METHOD M_AddChild : ERRORID
VAR_INPUT
	pObject : POINTER TO FB_Object;
	nSlotNr	: UINT;
	nIndex 	: INT;
END_VAR
//Der Delodot-Dispenser kann folgende Objekt-Typen aufnehmen
//Camera, Exposure, Nozzle
IF pObject > 0 THEN
	IF pObject^.P_eObjectType = E_ObjectType.OBJECTTYPE_Camera OR
		pObject^.P_eObjectType = E_ObjectType.OBJECTTYPE_Exposure OR
		pObject^.P_eObjectType = E_ObjectType.OBJECTTYPE_DummyTool OR
		pObject^.P_eObjectType = E_ObjectType.OBJECTTYPE_Nozzle THEN
		M_AddChild := SUPER^.M_AddChild(pObject,nSlotNr,nIndex);
	ELSE
		M_AddChild := E_ErrorIdObjMgmt.ERRORID_InvalidParentObject;
	END_IF
ELSE
	M_AddChild := E_ErrorIdObjMgmt.ERRORID_InvalidParentObject;
END_IF
END_METHOD

METHOD M_CancelAction
VAR_INPUT
	eAction : E_Action;
END_VAR
CASE eAction OF
	E_Action.ACTION_SetPressure:
		IF bSetPress  THEN
			fbSetPress(bExecute:= FALSE, pPneuChannelRef:= pPneuChannelPress);
		END_IF	
	E_Action.ACTION_SwitchPressure:
		IF bSwitchPress AND nStateA_SwitchPress < 70 THEN
			nStateA_SwitchPress := 70;
		END_IF
	E_Action.ACTION_DispenseDrops:
		IF bDispense AND nStateA_Dispense < 70 THEN
			nStateA_Dispense := 70;
		END_IF
ELSE
	SUPER^.M_CancelAction(eAction);
END_CASE
END_METHOD

METHOD M_CheckAction : ERRORID
VAR_INPUT
	refActionData 	: REFERENCE TO ST_ActionData;
	pCorrelObject	: POINTER TO FB_Object;
END_VAR

VAR
END_VAR
CASE refActionData.eAction OF
	E_Action.ACTION_DispenseDrops, //BasicAction für ActionOnArray
	E_Action.ACTION_TeachTarget:
		RETURN;
ELSE
	M_CheckAction := SUPER^.M_CheckAction(refActionData, pCorrelObject);
END_CASE
END_METHOD

METHOD M_CheckProcDataType : BOOL
VAR_INPUT
	eProcDataType : E_ProcDataType;
END_VAR
IF eProcDataType = E_ProcDataType.PROCDATATYPE_Temp1 THEN
	M_CheckProcDataType := TRUE;
END_IF
END_METHOD

METHOD M_ClearAllProps
VAR_INPUT
	bIgnoreParent : BOOL; //Es wird das gesamte OD gelöscht. -> Zeiger auf Parent nicht mehr gültig!
END_VAR
pPneuChannelPress := 0;
SUPER^.M_ClearAllProps(bIgnoreParent);
END_METHOD

METHOD M_ExeAction : ERRORID
VAR_INPUT
	refActionData : REFERENCE TO ST_ActionData;	
END_VAR
IF NOT (eCurrentState = E_MachineState.MACHINESTATE_Idle OR
	eCurrentState = E_MachineState.MACHINESTATE_Active OR
	eCurrentState = E_MachineState.MACHINESTATE_Ready) THEN
	M_ExeAction := E_ErrorIdCmd.ERRORID_InvalidState;
	RETURN;
END_IF

CASE refActionData.eAction OF
	
	E_Action.ACTION_Init:
		IF NOT bInitAxis AND NOT bInitTool THEN
			bInitAxis := TRUE;
			bInitTool := TRUE;
			fbList.A_AddHeadValue(hList:= hList, putValue := E_Action.ACTION_Init);	//InitAxis
			fbList.A_AddHeadValue(hList:= hList, putValue := E_Action.ACTION_Init);	//InitTool
		ELSE
			RETURN;
		END_IF
		
	E_Action.ACTION_SetPressure:
		fbSetPress(bExecute:= FALSE, pPneuChannelRef:= pPneuChannelPress); //eventueller Fehler wird auch zurückgesetzt
		fbSetPress.bAwait := DINT_TO_BOOL(refActionData.aParams[1]);
		fbSetPress.nValue := DINT_TO_INT(refActionData.aParams[2]);
		fbSetPress.nTolerancePlus := DINT_TO_INT(refActionData.aParams[3]);
		fbSetPress.nToleranceMinus := DINT_TO_INT(refActionData.aParams[4]);
		fbSetPress.tTimeout := DINT_TO_TIME(refActionData.aParams[5]);
		
		fbSetPress(bExecute:= TRUE,	pPneuChannelRef:= pPneuChannelPress,nErrorId=> M_ExeAction);
		IF fbSetPress.bError THEN
			RETURN;
		END_IF
		
		IF NOT bSetPress AND fbSetPress.bBusy THEN
			bSetPress := TRUE;
			fbList.A_AddHeadValue(hList := hList, putValue := E_Action.ACTION_SetPressure);
		ELSE
			RETURN;	
		END_IF

	E_Action.ACTION_SwitchPressure:
		eSwitchPressCtrl := DINT_TO_USINT(refActionData.aParams[1]);
		IF (eSwitchPressCtrl = E_PressCtrl.PRESSCTRL_PressOn) OR (eSwitchPressCtrl = E_PressCtrl.PRESSCTRL_Off) THEN
			tPressTime := DINT_TO_TIME(refActionData.aParams[2]);
			//Wenn Aktion aktiv kann es sein das die Zeit noch läuft oder der Druck an ist
			IF bSwitchPress THEN	//Aktion ist aktiv
				IF eSwitchPressCtrl = E_PressCtrl.PRESSCTRL_PressOn THEN
					//Statemachine zurücksetzen
					nStateA_SwitchPress := 0;		
				ELSE
					pFbMultiZ^.M_SetDigiOut(nChannel:= nDOutChanValvePress, bValue:= FALSE);
					nStateA_SwitchPress := 80;
				END_IF
			ELSE	//Aktion ist nicht aktiv
				IF eSwitchPressCtrl = E_PressCtrl.PRESSCTRL_PressOn THEN
					bSwitchPress := TRUE;
					fbList.A_AddHeadValue(hList := hList, putValue := E_Action.ACTION_SwitchPressure);
				ELSE
					pFbMultiZ^.M_SetDigiOut(nChannel:= nDOutChanValvePress, bValue:= FALSE);
				END_IF
			END_IF
		ELSE
			M_ExeAction := E_ErrorIdCmd.ERRORID_InvalidCtrl;
			RETURN;
		END_IF		
		
	E_Action.ACTION_DispenseDrops:
		bDispenseStart := DINT_TO_BOOL(refActionData.aParams[2]);
		IF NOT bDispense AND bDispenseStart THEN
			nDrops := DINT_TO_UINT(refActionData.aParams[1]);
			fbList.A_AddHeadValue( hList := hList, putValue := E_Action.ACTION_DispenseDrops);
			bDispense := TRUE;
		ELSE
			pTripleTrigRef^.M_TriggerOff(nTriggerChannel);
		END_IF

	ELSE
		M_ExeAction := SUPER^.M_ExeAction(refActionData);
		RETURN;
END_CASE
bBusy := TRUE;
eCurrentState := E_MachineState.MACHINESTATE_Active;
END_METHOD

METHOD M_GetAllProps : ERRORID
VAR_INPUT
	refCmdData : REFERENCE TO  ST_CmdData;
END_VAR
//BaseProperties lesen
SUPER^.M_GetAllProps(refCmdData);
//BaseProperties lesen
nCurrentPropIndex := nCurrentPropIndex + 1; //SubType (Reserve)
refCmdData.n32Data[nCurrentPropIndex] := nSubType;
nCurrentPropIndex := nCurrentPropIndex + 1;
refCmdData.n32Data[nCurrentPropIndex] := nTriggerChannel;
IF pTripleTrigRef > 0 THEN
	nCurrentPropIndex := nCurrentPropIndex + 1;
	refCmdData.n32Data[nCurrentPropIndex] := pTripleTrigRef^.M_GetFrequency(nTriggerChannel);
	nCurrentPropIndex := nCurrentPropIndex + 1;
	refCmdData.n32Data[nCurrentPropIndex] := pTripleTrigRef^.M_GetPulse(nTriggerChannel);
	nCurrentPropIndex := nCurrentPropIndex + 1;
	refCmdData.n32Data[nCurrentPropIndex] := pTripleTrigRef^.M_GetAmplitudePercent(nTriggerChannel);
ELSE
	nCurrentPropIndex := nCurrentPropIndex + 3;
END_IF
nCurrentPropIndex := nCurrentPropIndex + 1;
IF pPneuChannelPress > 0 THEN
	refCmdData.n32Data[nCurrentPropIndex] := pPneuChannelPress^.nChannel;
ELSE
	refCmdData.n32Data[nCurrentPropIndex] := 0;
END_IF
nCurrentPropIndex := nCurrentPropIndex + 1; 
refCmdData.n32Data[nCurrentPropIndex] := nDOutChanValvePress; //Digitaler Ausgangskanal MzHead Druckventil
END_METHOD

METHOD M_SetAllProps : ERRORID
VAR_INPUT
	refCmdData : REFERENCE TO  ST_CmdData;
END_VAR

VAR
	nPneuChannel : USINT;
END_VAR
M_SetAllProps := SUPER^.M_SetAllProps(refCmdData);

IF M_SetAllProps > 0 THEN
	RETURN;
END_IF

{IF defined (variable:aFbTripleTriggerRef)}
pTripleTrigRef := ADR(aFbTripleTriggerRef[1]);
{ELSE}
M_SetAllProps := E_ErrorIdObjMgmt.ERRORID_InvalidHardwareRef;
RETURN;
{END_IF}

//SubType (Reserve)
nCurrentPropIndex := nCurrentPropIndex + 1;
nSubType := refCmdData.n32Data[nCurrentPropIndex];
//TriggerChannel
nCurrentPropIndex := nCurrentPropIndex + 1;
nSpecPropIndex := nCurrentPropIndex;
nTriggerChannel := DINT_TO_USINT(refCmdData.n32Data[nCurrentPropIndex]);
IF NOT (nTriggerChannel >= 1 AND nTriggerChannel <= 3) THEN
	M_SetAllProps := E_ErrorIdObjMgmt.ERRORID_InvalidTriggerChannel;
	RETURN;
END_IF

//Frequenz
nCurrentPropIndex := nCurrentPropIndex + 1;
IF NOT (refCmdData.n32Data[nCurrentPropIndex] >= 16 AND refCmdData.n32Data[nCurrentPropIndex] <= 1000000) THEN	
	M_SetAllProps := E_ErrorIdObjMgmt.ERRORID_InvalidFrequency;
	RETURN;
END_IF
pTripleTrigRef^.M_SetFrequency(nTriggerChannel,refCmdData.n32Data[nCurrentPropIndex]);

//Plusbreite
nCurrentPropIndex := nCurrentPropIndex + 1;
IF NOT (refCmdData.n32Data[nCurrentPropIndex] >= 0 AND refCmdData.n32Data[nCurrentPropIndex] <= 65535) THEN
	M_SetAllProps := E_ErrorIdObjMgmt.ERRORID_InvalidPulseWidth;  //Error
	RETURN;
END_IF
pTripleTrigRef^.M_SetPulse(nTriggerChannel,DINT_TO_UINT(refCmdData.n32Data[nCurrentPropIndex]));

//Stroke(Hub) in % (1 Stelle hinter Komma)
nCurrentPropIndex := nCurrentPropIndex + 1;
IF NOT (refCmdData.n32Data[nCurrentPropIndex] >= 0 AND refCmdData.n32Data[nCurrentPropIndex] <= 1000) THEN
	M_SetAllProps := E_ErrorIdObjMgmt.ERRORID_InvalidVoltage;  //Error
	RETURN;
END_IF
pTripleTrigRef^.M_SetAmplitudePercent(nTriggerChannel,DINT_TO_UINT(refCmdData.n32Data[nCurrentPropIndex]));

//PneuChannel Druck
nCurrentPropIndex := nCurrentPropIndex + 1;
nPneuChannel := DINT_TO_USINT(refCmdData.n32Data[nCurrentPropIndex]);
IF NOT (nPneuChannel >= 0 AND nPneuChannel <= cNoOfPneuChannels) THEN
	M_SetAllProps := E_ErrorIdObjMgmt.ERRORID_InvalidPneuChannel;
	RETURN;	
END_IF
pPneuChannelPress := ADR(aFbPneuChannel[nPneuChannel]);

//Digitale Ausgänge auf MzHead müssen zwischen 1 und 7 liegen
nCurrentPropIndex := nCurrentPropIndex + 1;
nDOutChanValvePress := DINT_TO_USINT(refCmdData.n32Data[nCurrentPropIndex]);	//Digitaler Ausgangskanal MzHead Druckventil
IF NOT (nDOutChanValvePress >= 0 AND nDOutChanValvePress <= 7) THEN
	M_SetAllProps := E_ErrorIdObjMgmt.ERRORID_InvalidMzDOutChannel;
	RETURN;	
END_IF

nNoOfProps := nCurrentPropIndex + 1;
END_METHOD

METHOD M_SetSingleProp : ERRORID
VAR_INPUT
	refCmdData : REFERENCE TO  ST_CmdData;
END_VAR
IF nSpecPropIndex = refCmdData.aHeader[1] THEN
	IF refCmdData.n32Data[0] >= 1 AND refCmdData.n32Data[0] <= 3 THEN
		nTriggerChannel := DINT_TO_USINT(refCmdData.n32Data[0]);
	ELSE
		M_SetSingleProp := E_ErrorIdObjMgmt.ERRORID_InvalidTriggerChannel;
		RETURN;
	END_IF
ELSIF (nSpecPropIndex + 1) = refCmdData.aHeader[1] THEN	//Frequenz
	IF NOT (refCmdData.n32Data[0] > 16 AND refCmdData.n32Data[0] < 1000000) THEN
		M_SetSingleProp := E_ErrorIdObjMgmt.ERRORID_InvalidFrequency;
		RETURN;
	END_IF
	pTripleTrigRef^.M_SetFrequency(nTriggerChannel,refCmdData.n32Data[0]);
ELSIF (nSpecPropIndex + 2) = refCmdData.aHeader[1] THEN //Pulsbreite
	IF NOT (refCmdData.n32Data[0] >= 0 AND refCmdData.n32Data[0] < 65535) THEN
		M_SetSingleProp := E_ErrorIdObjMgmt.ERRORID_InvalidPulseWidth;
		RETURN;
	END_IF
	pTripleTrigRef^.M_SetPulse(nTriggerChannel,DINT_TO_UINT(refCmdData.n32Data[0]));
ELSIF (nSpecPropIndex + 3) = refCmdData.aHeader[1] THEN	//Stroke(Hub) in % (1 Stelle hinter Komma)
	IF NOT (refCmdData.n32Data[0] >= 0 AND refCmdData.n32Data[0] <= 1000) THEN
		M_SetSingleProp := E_ErrorIdObjMgmt.ERRORID_InvalidVoltage;
		RETURN;
	END_IF
	pTripleTrigRef^.M_SetAmplitudePercent(nTriggerChannel,DINT_TO_UINT(refCmdData.n32Data[0]));
ELSE
	M_SetSingleProp := SUPER^.M_SetSingleProp(refCmdData);
END_IF
END_METHOD

END_FUNCTION_BLOCK

// ---- Objects/Tools/FB_TriplePip.TcPOU
FUNCTION_BLOCK FB_TriplePip EXTENDS FB_MzTool
VAR_INPUT
END_VAR
VAR_OUTPUT
END_VAR
VAR
	bTipEjectorExist	: BOOL;	

	//SpecProperties
	nDiluterObjId		: UINT;
	pDiluter			: POINTER TO FB_Diluter;
	
	pPneuChannelSynthGas: POINTER TO FB_PneuChannelRef;
	pPneuChannelVac		: POINTER TO FB_PneuChannelRef;
	
	nValveNrSynthGas	: USINT;
	nValveNrVacuum		: USINT;
	nHoldVacuumVial		: INT;
	nHoldVacuumSeptum	: INT;
	rDockOffset			: REAL;
	rXMoveDockFlipTube	: REAL;
	rZMoveDockFlipTube	: REAL;

	//****************************************Aktionvariablen****************************************************
	
	stActionDataSpec	: ST_ActionData;
	
	//Action: "InitSpec"
	bInitSpec			: BOOL;
	bInitSpecFlag		: BOOL := TRUE;
	nStateA_InitSpec	: USINT;
	
	//Action: "Dispense"
	bDispense			: BOOL;
	nStateA_Dispense	: USINT;
	nQuantity			: DINT;
	nFlow				: DINT;
	
	//Action: "SetPressure"
	bSetPress			: BOOL;
	fbSetPress			: FB_SetPressure;

	//Action: "SetVacuum"
	bSetVacuum			: BOOL;
	fbSetVacuum			: FB_SetPressure;
	
	//Action: "SwitchPressure"
	bSwitchPress		: BOOL;			
	nStateA_SwitchPress	: USINT;		//State von A_SwitchPress()
	nSwitchPressChannel	: USINT;
	eSwitchPressCtrl	: E_PressCtrl;
	tPressTime			: TIME;			//nach dieser Zeit Ventil automatisch wieder zu
	timerPress			: TON;			//Timer für Öffnungszeit Druckventil 		
	
END_VAR

IF eCurrentState = E_MachineState.MACHINESTATE_Active THEN
	IF bInitSpec THEN
		A_InitSpec();
		IF nStateA_InitSpec >= 80 THEN
			IF nStateA_InitSpec >= 99 THEN
				bError := TRUE;		
			END_IF
			bInitSpec := FALSE;
			nStateA_InitSpec := 0;
			M_RemoveListEntry(nSearchValue:= E_Action.ACTION_Init);
		END_IF		
	END_IF
	
	IF bDispense THEN
		A_Dispense();
		IF nStateA_Dispense >= 80 THEN
			IF nStateA_Dispense >= 99 THEN
				bError := TRUE;	
			END_IF
			bDispense := FALSE;
			nStateA_Dispense := 0;
			M_RemoveListEntry(nSearchValue:= E_Action.ACTION_Dispense);
		END_IF
	END_IF
	
	IF bSetPress THEN
		fbSetPress(pPneuChannelRef:= pPneuChannelSynthGas);
		IF NOT fbSetPress.bBusy THEN
			IF fbSetPress.bError THEN
				bError := TRUE;
				stError.ErrorId := fbSetPress.nErrorId;
				stError.POU := E_POU.POU_FB_TriplePip;
				fbErrorList.M_Add(stError);
			END_IF
			bSetPress := FALSE;
			fbSetPress(pPneuChannelRef:= pPneuChannelSynthGas, bExecute:= FALSE);
			M_RemoveListEntry(nSearchValue:= E_Action.ACTION_SetPressure);
		END_IF
	END_IF	

	IF bSetVacuum THEN
		fbSetVacuum(pPneuChannelRef:= pPneuChannelVac);
		IF NOT fbSetVacuum.bBusy THEN
			IF fbSetVacuum.bError THEN
				bError := TRUE;
				stError.ErrorId := fbSetVacuum.nErrorId;
				stError.POU := E_POU.POU_FB_TriplePip;
				fbErrorList.M_Add(stError);
			END_IF
			bSetVacuum := FALSE;
			fbSetVacuum(pPneuChannelRef:= pPneuChannelVac, bExecute:= FALSE);
			M_RemoveListEntry(nSearchValue:= E_Action.ACTION_SetVacuum);
		END_IF
	END_IF	
	
	IF bSwitchPress THEN	//Kartuschendruck einstellen und Ein-bzw. Aus schalten 
		A_SwitchPress();
		IF nStateA_SwitchPress >= 80 THEN
			IF nStateA_SwitchPress >= 99 THEN
				bError := TRUE;
			END_IF
			bSwitchPress := FALSE;
			nStateA_SwitchPress := 0;
			M_RemoveListEntry(nSearchValue:= E_Action.ACTION_SwitchPressure);
		END_IF
	END_IF	
END_IF

SUPER^();	//FB_MzTool aufrufen

//Prozessdaten aktualisieren
IF pPneuChannelSynthGas > 0 THEN
	stProcessData.n32Data[7] := pPneuChannelSynthGas^.P_nCurrentPressure;
END_IF

IF pPneuChannelVac > 0 THEN
	stProcessData.n32Data[8] := pPneuChannelVac^.P_nCurrentPressure;
END_IF

IF nValveNrSynthGas > 0 THEN
	IF aValves[nValveNrSynthGas].bDigiOut1 THEN
		stProcessData.n32Data[9] := E_PressCtrl.PRESSCTRL_PressOn;
	ELSE
		stProcessData.n32Data[9] := E_PressCtrl.PRESSCTRL_Off;
	END_IF
END_IF

IF nValveNrVacuum > 0 THEN
	IF aValves[nValveNrVacuum].bDigiOut1 THEN
		stProcessData.n32Data[10] := E_PressCtrl.PRESSCTRL_VacOn;
	ELSE
		stProcessData.n32Data[10] := E_PressCtrl.PRESSCTRL_Off;
	END_IF
END_IF

aObjProcData[nNotifyId] := stProcessData;

ACTION A_Dispense:
IF pDiluter^.P_bError THEN
	stError.ErrorId := pDiluter^.P_nErrorId;
	stError.POUState := nStateA_Dispense;
	nStateA_Dispense := 99;
END_IF

CASE nStateA_Dispense OF
	0:	MEMSET(ADR(stActionDataSpec),0,SIZEOF(stActionDataSpec));
		//stActionDataSpec.bIntern := TRUE;
		stActionDataSpec.eAction := E_Action.ACTION_DilPump;
		stActionDataSpec.aParams[1] := E_DilPumpMode.MODE_Press;
		stActionDataSpec.aParams[2] := nQuantity; 
		stActionDataSpec.aParams[3] := nFlow;
		//stActionDataSpec.aParams[4] := 2000; //ReloadSpeed wird von DilConfig übernommen
		//stActionDataSpec.aParams[5] := 1; //Valve-Position für Pump
		//stActionDataSpec.aParams[6] := 2; //Valve-Position für Reload
		
		stError.ErrorId := pDiluter^.M_ExeAction(stActionDataSpec);
		IF stError.ErrorId > 0 THEN
			stError.POUState := nStateA_Dispense;
			nStateA_Dispense := 99;
		ELSE
			nStateA_Dispense := 1;	
		END_IF
		
	1:	//Warten bis Dispensierung fertig
		IF NOT pDiluter^.M_GetActionBusy(E_Action.ACTION_DilPump) THEN
			nStateA_Dispense := 80;
		END_IF
		
	70:	//Abbrechen
		MEMSET(ADR(stActionDataSpec),0,SIZEOF(stActionDataSpec));
		//stActionDataSpec.bIntern := TRUE;
		stActionDataSpec.eAction := E_Action.ACTION_Stop;
		
		pDiluter^.M_ExeAction(stActionDataSpec);
		nStateA_Dispense := 71;
		
	71:	
		IF NOT pDiluter^.P_bBusy THEN
			nStateA_Dispense := 80;
		END_IF
END_CASE

//Errorhandling
IF nStateA_Dispense = 99 THEN
	stError.Cmd := E_Action.ACTION_Dispense;
	stError.POU := E_POU.POU_FB_TriplePip;
	stError.POUAction := E_POUACT.POUACT_A_Dispense;
	fbErrorList.M_Add(stError);
END_IF
END_ACTION

ACTION A_InitSpec:
CASE nStateA_InitSpec OF
	0:	//Checken ob Diluter richtg zugeordnet
		
		IF fbObjectDirectory.M_GetObjType(nDiluterObjId) = E_ObjectType.OBJECTTYPE_Diluter THEN
			nStateA_InitSpec := 80;
		ELSE
			stError.ErrorId := E_ErrorIdObjMgmt.ERRORID_InvalidDiluterObjId;
			nStateA_InitSpec := 99;
		END_IF
	
	1:	//Checken ob notwendige Flüssigleiten vorhanden
	
	2:	//PCV-Level-Controlle aktivieren
	
END_CASE
END_ACTION

ACTION A_Reset:
//Ist noch eine Aktion aktiv?
IF nStateA_ResetSpec = 0 THEN 
	IF bDispense THEN
		bDispense := FALSE;
		nStateA_Dispense := 0;
	END_IF
	
	nStateA_ResetSpec := 80;
END_IF

SUPER^.A_Reset();
END_ACTION

ACTION A_Stop:
IF nStateA_Stop = 0 THEN

	IF bDispense AND nStateA_Dispense < 70 THEN
		nStateA_Dispense := 70;
	END_IF
	
	IF bSetPress THEN
		fbSetPress(bExecute:= FALSE, pPneuChannelRef:= pPneuChannelSynthGas);
	END_IF

	IF bSetVacuum THEN
		fbSetVacuum(bExecute:= FALSE, pPneuChannelRef:= pPneuChannelVac);
	END_IF
		
	
	nStateA_Stop := 1;
END_IF

SUPER^.A_Stop();
END_ACTION

ACTION A_SwitchPress:
CASE nStateA_SwitchPress OF
	0:	//Ventil Einschalten
		IF eSwitchPressCtrl = E_PressCtrl.PRESSCTRL_PressOn OR eSwitchPressCtrl = E_PressCtrl.PRESSCTRL_VacOn THEN
			aValves[M_GetValveNr(nSwitchPressChannel)].M_On(1);
		END_IF
	
		//Timer starten
		IF tPressTime = T#0S THEN
			nStateA_SwitchPress := 80;
			RETURN;	
		END_IF
		
		timerPress(IN:= FALSE);
		timerPress(IN:= TRUE, PT:= tPressTime);
		nStateA_SwitchPress := 1;
		
	1:	//Warten bis Zeitabgelaufen
		timerPress();
		IF timerPress.Q THEN
			timerPress(IN:= FALSE);
			aValves[M_GetValveNr(nSwitchPressChannel)].M_Off();
			nStateA_SwitchPress := 80;
		END_IF
		
	70:	//Abbrechen
		timerPress(IN:= FALSE);
		aValves[M_GetValveNr(nSwitchPressChannel)].M_Off();
		nStateA_SwitchPress := 80;
END_CASE
END_ACTION

METHOD FB_init : BOOL
VAR_INPUT
	bInitRetains : BOOL; // if TRUE, the retain variables are initialized (warm start / cold start)
	bInCopyCode : BOOL;  // if TRUE, the instance afterwards gets moved into the copy code (online change)
END_VAR
eObjectType := E_ObjectType.OBJECTTYPE_TriplePip;
eObjectGroup := E_ObjectGroup.OBJECTGROUP_MzTool OR E_ObjectGroup.OBJECTGROUP_Device;
END_METHOD

METHOD M_AddChild : ERRORID
VAR_INPUT
	pObject : POINTER TO FB_Object;
	nSlotNr	: UINT;
	nIndex 	: INT;
END_VAR
//Kann folgende Objekt-Typen aufnehmen
//Vial
IF pObject > 0 THEN
	IF pObject^.P_eObjectType = E_ObjectType.OBJECTTYPE_Vial THEN
		M_AddChild := SUPER^.M_AddChild(pObject,nSlotNr,nIndex);
	ELSE
		M_AddChild := E_ErrorIdObjMgmt.ERRORID_InvalidParentObject;
	END_IF
ELSE
	M_AddChild := E_ErrorIdObjMgmt.ERRORID_InvalidParentObject;
END_IF
END_METHOD

METHOD M_CancelAction
VAR_INPUT
	eAction : E_Action;
END_VAR
CASE eAction OF
	E_Action.ACTION_Dispense:
		IF bDispense AND nStateA_Dispense < 70 THEN
			nStateA_Dispense := 70;
		END_IF
		
	E_Action.ACTION_SetPressure:
		IF bSetPress THEN
			fbSetPress(bExecute:= FALSE, pPneuChannelRef:= pPneuChannelSynthGas);
		END_IF
	
	E_Action.ACTION_SetVacuum:
		IF bSetVacuum THEN
			fbSetVacuum(bExecute:= FALSE, pPneuChannelRef:= pPneuChannelVac);
		END_IF
		
	E_Action.ACTION_SwitchPressure:
		IF bSwitchPress AND nStateA_SwitchPress < 70 THEN
			nStateA_SwitchPress := 70;
		END_IF	
ELSE
	SUPER^.M_CancelAction(eAction);
END_CASE
END_METHOD

METHOD M_CheckAction : ERRORID
VAR_INPUT
	refActionData 	: REFERENCE TO ST_ActionData;
	pCorrelObject	: POINTER TO FB_Object;
END_VAR

VAR
	pRack : POINTER TO FB_Rack;
	pReactor : POINTER TO FB_Reactor;
	pSlot : POINTER TO FB_PieceSlot;
	pTarget : POINTER TO FB_TargetBase;
END_VAR
CASE refActionData.eAction OF
	E_Action.ACTION_ExchangePiece:
		pTarget := fbObjectDirectory.M_GetObjPointer(refActionData.nTarget);
		//Welches Piece soll gehandelt werden?
		IF refActionData.aParams[2] = 0 THEN //Drop
			IF pPiece = 0 THEN
				M_CheckAction := E_ErrorIdCmd.ERRORID_NoPieceOnTool;
				RETURN;	
			END_IF
			//TripePip kann folgende Pieces handeln
			//Vial, Septum
			IF pPiece^.P_eObjectType = E_ObjectType.OBJECTTYPE_Vial THEN
				//Target muss VialRack oder Reaktor sein
				IF pTarget^.P_eObjectType = E_ObjectType.OBJECTTYPE_VialRack THEN
					pRack := pTarget;
					//Slot muss frei sein
					pSlot := pRack^.M_GetSlot(DINT_TO_UINT(refActionData.aParams[1]));
					IF pSlot = 0 THEN
						M_CheckAction := E_ErrorIdCmd.ERRORID_InvalidTargetSlot;
						RETURN;
					ELSIF pSlot^.P_pPiece > 0 THEN
						M_CheckAction := E_ErrorIdCmd.ERRORID_PieceAlreadyInSlot;
						RETURN;
					END_IF
				ELSIF pTarget^.P_eObjectType = E_ObjectType.OBJECTTYPE_Reactor THEN
					//Slot muss frei sein
					//Hier kann ein Vial geholt werden
					pReactor := pTarget;
					IF pReactor^.P_pVial > 0 THEN
						M_CheckAction := E_ErrorIdCmd.ERRORID_PieceAlreadyInSlot;
						RETURN;
					END_IF
				ELSE
					M_CheckAction := E_ErrorIdCmd.ERRORID_UnsuitableTarget;
					RETURN;
				END_IF
			ELSIF pPiece^.P_eObjectType = E_ObjectType.OBJECTTYPE_Septum THEN
				//Target kann nur Reaktor mit Vial sein
				//Ob ein Vial im Reaktor steht, wird in FB_Reactor.M_CheckActon() geprüft 
				IF pTarget^.P_eObjectType <> E_ObjectType.OBJECTTYPE_Reactor THEN 
					M_CheckAction := E_ErrorIdCmd.ERRORID_UnsuitableTarget;
					RETURN;
				END_IF
			ELSE
				M_CheckAction := E_ErrorIdCmd.ERRORID_InvalidPieceType;
				RETURN;
			END_IF
		ELSE  //Take
			//Schon ein Piece am Tool?
			IF THIS^.pPiece > 0 THEN
				M_CheckAction := E_ErrorIdCmd.ERRORID_PieceAlreadyOnTool;
				RETURN;
			END_IF
			
			IF pTarget^.P_eObjectType = E_ObjectType.OBJECTTYPE_Reactor THEN
				//Hier kann ein Vial geholt werden
				pReactor := pTarget;
				IF pReactor^.P_pVial = 0 THEN
					M_CheckAction := E_ErrorIdCmd.ERRORID_NoPieceInSlot;
					RETURN;
				ELSIF pReactor^.P_pVial^.P_pSeptum > 0 THEN
					M_CheckAction := E_ErrorIdCmd.ERRORID_SeptumAlreadyOnVial;
					RETURN;
				END_IF
			ELSIF pTarget^.P_eObjectType = E_ObjectType.OBJECTTYPE_VialRack THEN
				//Hier kann ein Vial geholt werden
				pRack := pTarget;
				pSlot := pRack^.M_GetSlot(DINT_TO_UINT(refActionData.aParams[1]));
				IF pSlot > 0 THEN
					IF pSlot^.P_pPiece = 0 THEN
						M_CheckAction := E_ErrorIdCmd.ERRORID_NoPieceInSlot;
						RETURN;
					ELSIF pSlot^.P_pPiece^.P_eObjectType <> E_ObjectType.OBJECTTYPE_Vial THEN
						M_CheckAction := E_ErrorIdCmd.ERRORID_InvalidPieceType;
						RETURN;
					END_IF
				ELSE
					M_CheckAction := E_ErrorIdCmd.ERRORID_InvalidTargetSlot;
					RETURN;				
				END_IF		
			ELSIF pTarget^.P_eObjectType = E_ObjectType.OBJECTTYPE_SeptumRack THEN
				//Hier kann ein Septum geholt werden 
				pRack := pTarget;
				pSlot := pRack^.M_GetSlot(DINT_TO_UINT(refActionData.aParams[1]));
				IF pSlot > 0 THEN
					IF pSlot^.P_pPiece = 0 THEN
						M_CheckAction := E_ErrorIdCmd.ERRORID_NoPieceInSlot;
						RETURN;
					ELSIF pSlot^.P_pPiece^.P_eObjectType <> E_ObjectType.OBJECTTYPE_Septum THEN
						M_CheckAction := E_ErrorIdCmd.ERRORID_InvalidPieceType;
						RETURN;
					END_IF
				ELSE
					M_CheckAction := E_ErrorIdCmd.ERRORID_InvalidTargetSlot;
					RETURN;				
				END_IF
			END_IF
		END_IF
	E_Action.ACTION_DockTool:
		pTarget := fbObjectDirectory.M_GetObjPointer(refActionData.nTarget);
		//TripePip kann nur an den Reaktor, geschlossenes VialRack oder FlipTubeRack andocken
		IF pTarget^.P_eObjectType <> E_ObjectType.OBJECTTYPE_Reactor AND 
			pTarget^.P_eObjectType <> E_ObjectType.OBJECTTYPE_VialRackClosed AND
			pTarget^.P_eObjectType <> E_ObjectType.OBJECTTYPE_FlipTubeRack THEN
			M_CheckAction := E_ErrorIdCmd.ERRORID_UnsuitableTarget;
			RETURN;
		END_IF			
		//Piece am Tool?
		IF THIS^.pPiece > 0 THEN
			M_CheckAction := E_ErrorIdCmd.ERRORID_PieceAlreadyOnTool;
			RETURN;
		END_IF
	E_Action.ACTION_WashTool:
		//Washmode checken
		IF refActionData.aParams[2] = E_WashMode.MODE_WashInside THEN
			M_CheckAction := M_CheckBottles();
		ELSIF refActionData.aParams[2] = E_WashMode.MODE_WashOutside THEN
			;
		ELSIF refActionData.aParams[2] = E_WashMode.MODE_WashInOutside THEN
			M_CheckAction := M_CheckBottles();
		ELSE
			M_CheckAction := E_ErrorIdCmd.ERRORID_InvalidWashMode;	
		END_IF
	E_Action.ACTION_TeachTarget:
		RETURN;
ELSE
	M_CheckAction := SUPER^.M_CheckAction(refActionData, pCorrelObject);
END_CASE
END_METHOD

METHOD M_CheckBottles : ERRORID
VAR_INPUT
END_VAR
IF pDiluter > 0 THEN
	M_CheckBottles := pDiluter^.M_CheckBottles(0);
END_IF
END_METHOD

METHOD M_CheckProps : ERRORID
VAR_INPUT
END_VAR
M_CheckProps := SUPER^.M_CheckProps();
IF M_CheckProps > 0 THEN
	RETURN;
END_IF

//Konfigurierte Properties checken
//zugeordneter Diuter
IF fbObjectDirectory.M_GetObjType(nDiluterObjId) <> E_ObjectType.OBJECTTYPE_Diluter THEN
	M_CheckProps := E_ErrorIdObjMgmt.ERRORID_InvalidDiluterObjId; //Error
	RETURN;
ELSE
	pDiluter := fbObjectDirectory.M_GetObjPointer(nDiluterObjId);
END_IF
END_METHOD

METHOD M_ClearAllProps
VAR_INPUT
	bIgnoreParent : BOOL; //Es wird das gesamte OD gelöscht. -> Zeiger auf Parent nicht mehr gültig!
END_VAR
pPneuChannelSynthGas := 0;
pPneuChannelVac := 0;
SUPER^.M_ClearAllProps(bIgnoreParent);
END_METHOD

METHOD M_ExeAction : ERRORID
VAR_INPUT
	refActionData : REFERENCE TO ST_ActionData;	
END_VAR
IF NOT (eCurrentState = E_MachineState.MACHINESTATE_Idle OR
	eCurrentState = E_MachineState.MACHINESTATE_Active OR
	eCurrentState = E_MachineState.MACHINESTATE_Ready) THEN
	M_ExeAction := E_ErrorIdCmd.ERRORID_InvalidState;
	RETURN;
END_IF

CASE refActionData.eAction OF
	
	E_Action.ACTION_Init:
		IF NOT bInitAxis AND NOT bInitSpec THEN
			bInitAxis := TRUE;
			bInitSpec := TRUE;
			fbList.A_AddHeadValue( hList := hList, putValue := E_Action.ACTION_Init);	//InitBase
			fbList.A_AddHeadValue( hList := hList, putValue := E_Action.ACTION_Init);	//InitSpec
			//bIsInit := FALSE;
		ELSE
			RETURN;
		END_IF
		
	E_Action.ACTION_Dispense:
		IF NOT bDispense THEN
			M_ExeAction := pDiluter^.M_CheckBottles(0); //Checken, ob Bottles OK
			IF M_ExeAction > 0 THEN
				RETURN;
			END_IF			
			nQuantity := refActionData.aParams[1];
			nFlow := refActionData.aParams[2];
			fbList.A_AddHeadValue(hList := hList, putValue := E_Action.ACTION_Dispense);
			bDispense := TRUE;
		END_IF
	
	E_Action.ACTION_SetPressure:
		fbSetPress(bExecute:= FALSE, pPneuChannelRef:= pPneuChannelSynthGas); //eventueller Fehler wird auch zurückgesetzt
		fbSetPress.bAwait := DINT_TO_BOOL(refActionData.aParams[1]);
		fbSetPress.nValue := DINT_TO_INT(refActionData.aParams[2]);
		fbSetPress.nTolerancePlus := DINT_TO_INT(refActionData.aParams[3]);
		fbSetPress.nToleranceMinus := DINT_TO_INT(refActionData.aParams[4]);
		fbSetPress.tTimeout := DINT_TO_TIME(refActionData.aParams[5]);
		
		fbSetPress(bExecute:= TRUE,	pPneuChannelRef:= pPneuChannelSynthGas, nErrorId=> M_ExeAction);
		IF fbSetPress.bError THEN
			RETURN;
		END_IF
		
		IF NOT bSetPress AND fbSetPress.bBusy THEN
			bSetPress := TRUE;
			fbList.A_AddHeadValue(hList := hList, putValue := E_Action.ACTION_SetPressure);
		ELSE
			RETURN;	
		END_IF

	E_Action.ACTION_SetVacuum:
		fbSetVacuum(bExecute:= FALSE, pPneuChannelRef:= pPneuChannelVac); //eventueller Fehler wird auch zurückgesetzt
		fbSetVacuum.bAwait := DINT_TO_BOOL(refActionData.aParams[1]);
		fbSetVacuum.nValue := DINT_TO_INT(refActionData.aParams[2]);
		fbSetVacuum.nTolerancePlus := DINT_TO_INT(refActionData.aParams[3]);
		fbSetVacuum.nToleranceMinus := DINT_TO_INT(refActionData.aParams[4]);
		fbSetVacuum.tTimeout := DINT_TO_TIME(refActionData.aParams[5]);
		
		fbSetVacuum(bExecute:= TRUE, pPneuChannelRef:= pPneuChannelVac, nErrorId=> M_ExeAction);
		IF fbSetVacuum.bError THEN
			RETURN;
		END_IF
		
		IF NOT bSetVacuum AND fbSetVacuum.bBusy THEN
			bSetVacuum := TRUE;
			fbList.A_AddHeadValue(hList := hList, putValue := E_Action.ACTION_SetVacuum);
		ELSE
			RETURN;	
		END_IF
		
	E_Action.ACTION_SwitchPressure:
		//Channel checken
		nSwitchPressChannel := DINT_TO_USINT(refActionData.aParams[1]);
		IF M_GetValveNr(nSwitchPressChannel) = 0 THEN
			M_ExeAction := E_ErrorIdObjMgmt.ERRORID_InvalidPneuChannel;
			RETURN;
		END_IF
		eSwitchPressCtrl := DINT_TO_USINT(refActionData.aParams[2]);
		tPressTime := DINT_TO_TIME(refActionData.aParams[3]);
		IF bSwitchPress THEN	//Aktion ist aktiv
			//Statemachine zurücksetzen
		 	nStateA_SwitchPress := 0;		
			aValves[M_GetValveNr(nSwitchPressChannel)].M_Off();
			nStateA_SwitchPress := 80;
		ELSE //Aktion ist nicht aktiv
			IF eSwitchPressCtrl = E_PressCtrl.PRESSCTRL_PressOn OR eSwitchPressCtrl = E_PressCtrl.PRESSCTRL_VacOn THEN
				bSwitchPress := TRUE;
				fbList.A_AddHeadValue(hList := hList, putValue := E_Action.ACTION_SwitchPressure);
			ELSE
				aValves[M_GetValveNr(nSwitchPressChannel)].M_Off();
			END_IF			
		END_IF
	ELSE
		M_ExeAction := SUPER^.M_ExeAction(refActionData);
		RETURN;
END_CASE

bBusy := TRUE;
eCurrentState := E_MachineState.MACHINESTATE_Active;
END_METHOD

METHOD M_GetAllProps : ERRORID
VAR_INPUT
	refCmdData : REFERENCE TO  ST_CmdData;
END_VAR
//BaseProperties lesen
SUPER^.M_GetAllProps(refCmdData);
//BaseProperties lesen
nCurrentPropIndex := nCurrentPropIndex + 1;
refCmdData.n32Data[nCurrentPropIndex] := nDiluterObjId;

nCurrentPropIndex := nCurrentPropIndex + 1; 
IF pPneuChannelSynthGas > 0 THEN
	refCmdData.n32Data[nCurrentPropIndex] := pPneuChannelSynthGas^.nChannel;
ELSE
	refCmdData.n32Data[nCurrentPropIndex] := 0;
END_IF

nCurrentPropIndex := nCurrentPropIndex + 1;
IF pPneuChannelVac > 0 THEN
	refCmdData.n32Data[nCurrentPropIndex] := pPneuChannelVac^.nChannel;
ELSE
	refCmdData.n32Data[nCurrentPropIndex] := 0;
END_IF

nCurrentPropIndex := nCurrentPropIndex + 1;
refCmdData.n32Data[nCurrentPropIndex] := nValveNrSynthGas;
nCurrentPropIndex := nCurrentPropIndex + 1;
refCmdData.n32Data[nCurrentPropIndex] := nValveNrVacuum;
nCurrentPropIndex := nCurrentPropIndex + 1;
refCmdData.n32Data[nCurrentPropIndex] := nHoldVacuumVial;
nCurrentPropIndex := nCurrentPropIndex + 1;
refCmdData.n32Data[nCurrentPropIndex] := nHoldVacuumSeptum;
nCurrentPropIndex := nCurrentPropIndex + 1;
refCmdData.n32Data[nCurrentPropIndex] := REAL_TO_DINT(rDockOffset);
nCurrentPropIndex := nCurrentPropIndex + 1;
refCmdData.n32Data[nCurrentPropIndex] := REAL_TO_DINT(rXMoveDockFlipTube);
nCurrentPropIndex := nCurrentPropIndex + 1;
refCmdData.n32Data[nCurrentPropIndex] := REAL_TO_DINT(rZMoveDockFlipTube);
END_METHOD

METHOD M_GetVacuumOk : BOOL
VAR_INPUT
	nSetPressValue : INT;
	nSetPressTolPlus : INT;
	nSetPressTolMin : INT;
END_VAR
IF pPneuChannelVac > 0 THEN
	M_GetVacuumOk := pPneuChannelVac^.M_GetPressOk(nSetPressure:= nSetPressValue,nTolerancePlus:= nSetPressTolPlus, nToleranceMinus:= nSetPressTolMin);
END_IF
END_METHOD

METHOD PRIVATE M_GetValveNr : USINT
VAR_INPUT
	nChannel : USINT;
END_VAR
IF nChannel = 1 THEN
	M_GetValveNr := nValveNrSynthGas;
ELSIF nChannel = 2 THEN
	M_GetValveNr := nValveNrVacuum;
END_IF
END_METHOD

METHOD M_SetAllProps : ERRORID
VAR_INPUT
	refCmdData : REFERENCE TO  ST_CmdData;
END_VAR

VAR
	nPneuChannel : USINT;
END_VAR
M_SetAllProps := SUPER^.M_SetAllProps(refCmdData);

IF M_SetAllProps > 0 THEN
	RETURN;
END_IF

//Diluter
nCurrentPropIndex := nCurrentPropIndex + 1;
nSpecPropIndex := nCurrentPropIndex;
nDiluterObjId :=  DINT_TO_UINT(refCmdData.n32Data[nCurrentPropIndex]);
IF fbObjectDirectory.M_GetObjType(nDiluterObjId) = E_ObjectType.OBJECTTYPE_Diluter THEN
	pDiluter := fbObjectDirectory.M_GetObjPointer(nDiluterObjId);
ELSE
	M_SetAllProps := E_ErrorIdObjMgmt.ERRORID_InvalidDiluterObjId;
	RETURN;
END_IF

//PneuChannel Synthese-Gas
nCurrentPropIndex := nCurrentPropIndex + 1;
nPneuChannel := DINT_TO_USINT(refCmdData.n32Data[nCurrentPropIndex]);
IF NOT (nPneuChannel > 0 AND nPneuChannel <= cNoOfPneuChannels) THEN
	M_SetAllProps := E_ErrorIdObjMgmt.ERRORID_InvalidPneuChannel;
	RETURN;	
END_IF
pPneuChannelSynthGas := ADR(aFbPneuChannel[nPneuChannel]);

//PneuChannel Vakuum
nCurrentPropIndex := nCurrentPropIndex + 1;
nPneuChannel := DINT_TO_USINT(refCmdData.n32Data[nCurrentPropIndex]);		
IF NOT (nPneuChannel > 0 AND nPneuChannel <= cNoOfPneuChannels) THEN
	M_SetAllProps := E_ErrorIdObjMgmt.ERRORID_InvalidPneuChannel;
	RETURN;	
END_IF
pPneuChannelVac := ADR(aFbPneuChannel[nPneuChannel]);

nCurrentPropIndex := nCurrentPropIndex + 1;
nValveNrSynthGas := DINT_TO_USINT(refCmdData.n32Data[nCurrentPropIndex]);
IF NOT (nValveNrSynthGas > 0 AND nValveNrSynthGas <= cNoOfValves) THEN
	M_SetAllProps := E_ErrorIdObjMgmt.ERRORID_InvalidValveNumber;
	RETURN;
END_IF

nCurrentPropIndex := nCurrentPropIndex + 1;
nValveNrVacuum := DINT_TO_USINT(refCmdData.n32Data[nCurrentPropIndex]);
IF NOT (nValveNrVacuum > 0 AND nValveNrVacuum <= cNoOfValves) THEN
	M_SetAllProps := E_ErrorIdObjMgmt.ERRORID_InvalidValveNumber;
	RETURN;
END_IF

nCurrentPropIndex := nCurrentPropIndex + 1;
nHoldVacuumVial := DINT_TO_INT(refCmdData.n32Data[nCurrentPropIndex]);

nCurrentPropIndex := nCurrentPropIndex + 1;
nHoldVacuumSeptum := DINT_TO_INT(refCmdData.n32Data[nCurrentPropIndex]);

nCurrentPropIndex := nCurrentPropIndex + 1;
rDockOffset := DINT_TO_REAL(refCmdData.n32Data[nCurrentPropIndex]);

nCurrentPropIndex := nCurrentPropIndex + 1;
rXMoveDockFlipTube := DINT_TO_REAL(refCmdData.n32Data[nCurrentPropIndex]);

nCurrentPropIndex := nCurrentPropIndex + 1;
rZMoveDockFlipTube := DINT_TO_REAL(refCmdData.n32Data[nCurrentPropIndex]);

nNoOfProps := nCurrentPropIndex + 1;
END_METHOD

METHOD M_SetSingleProp : ERRORID
VAR_INPUT
	refCmdData : REFERENCE TO  ST_CmdData;
END_VAR

VAR
	nPneuChannel : USINT;
END_VAR
IF nSpecPropIndex + 1 = refCmdData.aHeader[1] THEN	//PneuChannelSynthGas
	nPneuChannel := DINT_TO_USINT(refCmdData.n32Data[0]);
	IF NOT (nPneuChannel > 0 AND nPneuChannel <= cNoOfPneuChannels) THEN
		M_SetSingleProp := E_ErrorIdObjMgmt.ERRORID_InvalidPneuChannel;
		RETURN;	
	END_IF
	pPneuChannelSynthGas := ADR(aFbPneuChannel[nPneuChannel]);
	
ELSIF nSpecPropIndex + 2 = refCmdData.aHeader[1] THEN	//PneuChannelVacuum
	nPneuChannel := DINT_TO_USINT(refCmdData.n32Data[0]);
	IF NOT (nPneuChannel > 0 AND nPneuChannel <= cNoOfPneuChannels) THEN
		M_SetSingleProp := E_ErrorIdObjMgmt.ERRORID_InvalidPneuChannel;
		RETURN;	
	END_IF
	pPneuChannelVac := ADR(aFbPneuChannel[nPneuChannel]);
	
ELSIF nSpecPropIndex + 3 = refCmdData.aHeader[1] THEN	//ValveSynthGas
	IF refCmdData.n32Data[0] >= 0 AND refCmdData.n32Data[0] <= cNoOfValves THEN
		nValveNrSynthGas := DINT_TO_USINT(refCmdData.n32Data[0]);
	ELSE
		M_SetSingleProp := E_ErrorIdObjMgmt.ERRORID_InvalidValveNumber;
	END_IF
	
ELSIF nSpecPropIndex + 4 = refCmdData.aHeader[1] THEN	//ValveNrVacuum
	IF refCmdData.n32Data[0] >= 0 AND refCmdData.n32Data[0] <= cNoOfValves THEN
		nValveNrVacuum := DINT_TO_USINT(refCmdData.n32Data[0]);
	ELSE
		M_SetSingleProp := E_ErrorIdObjMgmt.ERRORID_InvalidValveNumber;
	END_IF
	
ELSIF nSpecPropIndex + 5 = refCmdData.aHeader[1] THEN	//HoldVacVial
	nHoldVacuumVial := DINT_TO_INT(refCmdData.n32Data[0]);
ELSIF nSpecPropIndex + 6 = refCmdData.aHeader[1] THEN	//HoldVacSeptum
	nHoldVacuumSeptum := DINT_TO_INT(refCmdData.n32Data[0]);
ELSIF nSpecPropIndex + 7 = refCmdData.aHeader[1] THEN	//DockOffset
	rDockOffset := DINT_TO_REAL(refCmdData.n32Data[0]);
ELSIF nSpecPropIndex + 8 = refCmdData.aHeader[1] THEN	//XMoveDockFliptube
	rXMoveDockFlipTube := DINT_TO_REAL(refCmdData.n32Data[0]);
ELSIF nSpecPropIndex + 9 = refCmdData.aHeader[1] THEN	//ZMoveDockFliptube
	rZMoveDockFlipTube := DINT_TO_REAL(refCmdData.n32Data[0]);	
ELSE
	M_SetSingleProp := SUPER^.M_SetSingleProp(refCmdData);
END_IF
END_METHOD

PROPERTY P_nHoldVacSept : INT
GET
P_nHoldVacSept := nHoldVacuumSeptum;
END_GET
END_PROPERTY

PROPERTY P_nHoldVacVial : INT
GET
P_nHoldVacVial := nHoldVacuumVial;
END_GET
END_PROPERTY

PROPERTY P_rDockOffset : REAL
GET
P_rDockOffset := rDockOffset;
END_GET
END_PROPERTY

PROPERTY P_rXMoveDockFliptube : REAL
GET
P_rXMoveDockFliptube := rXMoveDockFlipTube;
END_GET
END_PROPERTY

PROPERTY P_rZMoveDockFliptube : REAL
GET
P_rZMoveDockFliptube := rZMoveDockFlipTube;
END_GET
END_PROPERTY

END_FUNCTION_BLOCK

// ---- Objects/Targets/Active/FB_Reactor.TcPOU
FUNCTION_BLOCK FB_Reactor EXTENDS FB_ActiveTarget IMPLEMENTS I_SlotTarget
VAR

	//Hardware-Verküpfung
	pDriveRef			: POINTER TO FB_HwRefReactDrive;
	pHeaterRef			: POINTER TO FB_HwRefReactHeater;
	
	nNoOfSlots			: USINT;
	fbVialSlot			: FB_PieceSlot(pOwner:= THIS);
	nValveNrCool		: USINT;	//VentilNr Kühlung (FBox)

	//Variablen allgemeine Statemachine
	
	//Process-Daten
	nTempActual			: UINT;
	
	//****************************************Aktionvariablen****************************************************
	bActionLock			: ARRAY[50..150] OF BOOL;

	fbReactDriveInit	: FB_ReactDriveInit;
	
	bDetectVial				: BOOL;
	nStateA_DetectVial		: USINT;
	nStateA_DetectVialNext	: USINT;
	eLastState				: E_OpClState;
	eEndState				: E_OpClState;
	
	//Action: "Heating"
	//bHeating			: BOOL;		//Action A_Heating() aktiv setzen
	nStateA_Heating		: USINT;	//State von A_Heating()
	nTempSetpoint		: USINT;	//SollTemperatur in °C
	bHeaterOn			: BOOL;

	//Action: "Cooling"
	bCooling			: BOOL;		//Action A_Cooling() aktiv setzen
	nStateA_Cooling		: USINT;	//State von A_Cooling()
	nTempCooling		: UINT;		//Bei Mtp-Holder bzw. SubstHolder in 10tel °C
	bCoolingOn			: BOOL;
	timerCooling		: TON;
	
	//Action: "OpenClose
	bOpenClose				: BOOL;
	nStateA_OpenClose		: USINT;
	nStateA_OpenCloseNext	: USINT;
	eReactComponent			: E_ReactDrive;
	eReactDrive				: E_ReactDrive;
	eOpClCtrl				: E_OpClCtrl;
	fbReactDriveMove		: FB_ReactDriveMove;
	nOpClPosition			: DINT;
		
END_VAR

IF bInitFB THEN
	bInitFB := FALSE;
	F_CreateLinkedListHnd( ADR( aNodes ), SIZEOF( aNodes ), hList );
	//Fehlerstruktur vorausfüllen
	stError.ObjectId := nObjectID;
	stError.HardwareGrp := E_HardwareGrp.Nothing;
	stError.POU := E_POU.POU_FB_Reactor;
END_IF

CASE eCurrentState OF
			
	E_MachineState.MACHINESTATE_Active:
		//BasicActions ausführen
		IF bInit THEN	//Initialisieren
			A_Init();
			IF nStateA_Init >= 80 THEN
				IF nStateA_Init >= 99 THEN
					bError := TRUE;
				END_IF
				bInit := FALSE;
				nStateA_Init := 0;
				M_RemoveListEntry(nSearchValue:= E_Action.ACTION_Init);
			END_IF
		END_IF
		
		IF bCooling THEN
			A_Cooling();
			IF nStateA_Cooling = 80 THEN
				bCooling := FALSE;
				nStateA_Cooling := 0;
				M_RemoveListEntry(nSearchValue:= E_Action.ACTION_Cooling);
				bBusy := FALSE;
			END_IF
		END_IF		
		
		IF bDetectVial THEN
			A_DetectVial();
			IF nStateA_DetectVial >= 80 THEN
				IF nStateA_DetectVial >= 99 THEN
					bError := TRUE;
				END_IF
				bDetectVial := FALSE;
				nStateA_DetectVial := 0;
				M_RemoveListEntry(nSearchValue:= E_Action.ACTION_DetectVial);
			END_IF
		END_IF
	
		IF bOpenClose THEN
			A_OpenClose();
			IF nStateA_OpenClose >= 80 THEN
				IF nStateA_OpenClose >= 99 THEN
					bError := TRUE;
				END_IF
				bOpenClose := FALSE;
				nStateA_OpenClose := 0;
				M_RemoveListEntry(nSearchValue:= E_Action.ACTION_ReactorOpCl);
			END_IF
		END_IF

		IF bStop THEN	//alle Actions stoppen
			A_Stop();
			IF nStateA_Stop >= 80 THEN
				IF nStateA_Stop >= 99 THEN
					bError := TRUE;
				END_IF
				bStop := FALSE;
				nStateA_Stop := 0;
				bCanceled := TRUE;
				M_RemoveListEntry(nSearchValue:= E_Action.ACTION_Stop);
			END_IF							
		END_IF

		IF hList.nCount = 0 THEN
			eCurrentState := E_MachineState.MACHINESTATE_Ready;
		END_IF

		IF bError  THEN
			eCurrentState := E_MachineState.MACHINESTATE_Error;
		END_IF

	E_MachineState.MACHINESTATE_Reset:
		A_Reset();
		IF nStateA_Reset = 80 THEN
			nStateA_Init := 0;
			nStateA_Stop := 0;
			nStateA_Reset := 0;
			bBusy := FALSE;
			bError := FALSE;
			bStopAllOnError := FALSE;
			fbList.A_Reset( hList := hList);
			MEMSET(ADR(bActionLock),0,SIZEOF(bActionLock));
			nErrorId := 0;
			stError.Cmd := 0;
			stError.ErrorId := 0;
			eCurrentState := E_MachineState.MACHINESTATE_Idle;
		ELSIF
			nStateA_Reset = 99 THEN
			fbErrorList.M_Add(stError);
			nStateA_Reset := 0;
			bBusy := FALSE;
			bError := TRUE;
			eCurrentState := E_MachineState.MACHINESTATE_Error;			
		END_IF

	E_MachineState.MACHINESTATE_Ready:
		bBusy := FALSE;
		eCurrentState := E_MachineState.MACHINESTATE_Idle;
	
	E_MachineState.MACHINESTATE_Error:
		bBusy := FALSE;
END_CASE


//Prozessdaten aktualisieren
stProcessData.nObjId := nObjectID;
stProcessData.n32Data[0] := BOOL_TO_DINT(bIsInit);
stProcessData.n32Data[1] := eCurrentState;
stProcessData.n32Data[2] := stError.ErrorId;
IF pHeaterRef > 0 THEN
nTempActual := pHeaterRef^.P_nTempActual;
stProcessData.n32Data[3] := BOOL_TO_DINT(pHeaterRef^.P_bHeatingOn);	
stProcessData.n32Data[4] := nTempActual;
END_IF

stProcessData.n32Data[5] := BOOL_TO_DINT(aValves[nValveNrCool].bDigiOut1);
stProcessData.n32Data[6] := pDriveRef^.eCurrentState[E_ReactDrive.Clamp];
stProcessData.n32Data[7] := pDriveRef^.eCurrentState[E_ReactDrive.CoverHoriz];
stProcessData.n32Data[8] := pDriveRef^.eCurrentState[E_ReactDrive.CoverVerti];
aObjProcData[nNotifyId] := stProcessData;

ACTION A_Cooling:
CASE nStateA_Cooling OF
	0:	aValves[nValveNrCool].M_On(1);
		nStateA_Cooling := 1;
		//Heizung ausschalten
		IF pHeaterRef > 0 THEN
			pHeaterRef^.P_bHeatingOn := FALSE;
		END_IF
					
	1:	//Warten bis Temp erreicht
		IF nTempActual <= nTempCooling THEN
			aValves[nValveNrCool].M_Off();
			nStateA_Cooling := 80;
		END_IF
		
	70:	//Abbrechen
		aValves[nValveNrCool].M_Off();
		nStateA_Cooling := 80;
END_CASE
END_ACTION

ACTION A_DetectVial:
CASE nStateA_DetectVial OF
	0:	//Klemme öffnen
		eLastState := pDriveRef^.eCurrentState[E_ReactDrive.Clamp];
		fbReactDriveMove.eOpClCtrl := E_OpClCtrl.Open;
		nStateA_DetectVial := 60;
		nStateA_DetectVialNext := 1;
		
	1:	//Sensor zurücksetzen
		pHeaterRef^.P_bResetVialDetect := TRUE;
		nStateA_DetectVial := 2;
	
	2:	//Klemme schließen
		pHeaterRef^.P_bResetVialDetect := FALSE;
		fbReactDriveMove.eOpClCtrl := E_OpClCtrl.Close;
		nStateA_DetectVial := 60;
		nStateA_DetectVialNext := 3;
	
	3:	//Wenn EndState "Open" dann wieder öffnen
		CASE eEndState OF
			E_OpClState.UNDEFINED:	//Wieder in den ursprüglichen State fahren
				IF eLastState = E_OpClState.Open THEN 
					fbReactDriveMove.eOpClCtrl := E_OpClCtrl.Open;
					nStateA_DetectVial := 60;
					nStateA_DetectVialNext := 80;
				ELSE
					nStateA_DetectVial := 80;	
				END_IF
			E_OpClState.Open:
				fbReactDriveMove.eOpClCtrl := E_OpClCtrl.Open;
				nStateA_DetectVialNext := 80;
				nStateA_DetectVial := 60;
			E_OpClState.Closed:
				fbReactDriveMove.eOpClCtrl := E_OpClCtrl.Close;
				nStateA_DetectVialNext := 80;
				nStateA_DetectVial := 60;
		END_CASE
END_CASE

IF nStateA_DetectVial = 60 THEN
	fbReactDriveMove(pDriveRef:= pDriveRef, eDrive:= E_ReactDrive.Clamp, bExecute:= TRUE); 
	IF NOT fbReactDriveMove.bBusy THEN
		IF fbReactDriveMove.bError THEN
			stError.ErrorId := fbReactDriveMove.nErrorId;
			stError.POUState := nStateA_DetectVial;
			nStateA_DetectVial := 99;
		ELSE
			nStateA_DetectVial := nStateA_DetectVialNext;
		END_IF
		fbReactDriveMove(bExecute:= FALSE);
	END_IF	
ELSIF nStateA_DetectVial = 70 THEN
	//Abbrechen
	;
END_IF

//Errorhandling
IF nStateA_DetectVial = 99 THEN
	stError.Cmd := E_Action.ACTION_DetectVial;
	stError.POUAction := E_POUACT.POUACT_A_DetectVial;
	fbErrorList.M_Add(stError);
END_IF
END_ACTION

ACTION A_Init:
IF nStateA_Init = 0 THEN
		bIsInit := FALSE;
		IF bFlagA_Init XOR fbReactDriveInit.bBusy  THEN
			bFlagA_Init := FALSE;
			fbReactDriveInit(pDriveRef := pDriveRef, bExecute:= TRUE);
		ELSE
			RETURN;
		END_IF
ELSIF nStateA_Init = 70 THEN //Abbrechen
	fbReactDriveInit.M_Stop();
	fbReactDriveInit();
END_IF		

IF NOT fbReactDriveInit.bBusy THEN
	IF fbReactDriveInit.bError THEN
		stError.ErrorId := fbReactDriveInit.nErrorId;
		stError.POUState := nStateA_Init;
		nStateA_Init := 99;
	ELSE
		IF nStateA_Init = 0 THEN
			bIsInit := TRUE;
		END_IF
		nStateA_Init := 80;
	END_IF
	fbReactDriveInit(pDriveRef := pDriveRef, bExecute:= FALSE);
	bFlagA_Init := TRUE;
END_IF

//Errorhandling
IF nStateA_Init = 99 THEN
	stError.Cmd := E_Action.ACTION_Init;
	stError.POUAction := E_POUACT.POUACT_A_Init;
	fbErrorList.M_Add(stError);
END_IF
END_ACTION

ACTION A_OpenClose:
IF nStateA_OpenClose <> 60 THEN
	stError.POUState := nStateA_OpenClose;
END_IF

CASE nStateA_OpenClose OF
	0:	//Auswahl, welche Komponenten
		fbReactDriveMove.eOpClCtrl := eOpClCtrl;
		CASE eReactComponent OF
			//Einzelne Komponenten
			E_ReactDrive.Clamp:
				eReactDrive := E_ReactDrive.Clamp;
				nStateA_OpenClose := 60;
				nStateA_OpenCloseNext := 80;
			E_ReactDrive.CoverHoriz:
				eReactDrive := E_ReactDrive.CoverHoriz;
				nStateA_OpenClose := 60;
				nStateA_OpenCloseNext := 80;
			E_ReactDrive.CoverVerti:
				eReactDrive := E_ReactDrive.CoverVerti;
				nStateA_OpenClose := 60;
				nStateA_OpenCloseNext := 80;
			E_ReactDrive.CoverBoth:
				IF eOpClCtrl = E_OpClCtrl.Open THEN
					nStateA_OpenClose := 1;	
				ELSE
					nStateA_OpenClose := 5;
				END_IF
			E_ReactDrive.Complete:
				IF eOpClCtrl = E_OpClCtrl.Open THEN
					nStateA_OpenClose := 10;	
				ELSE
					nStateA_OpenClose := 13;
				END_IF
		END_CASE
	
		///////////////////////////////CoverBoth open////////////////////////////////////////////
	1:	//Clamp schließen, um Vial zurückzuhalten
		eReactDrive := E_ReactDrive.Clamp;
		fbReactDriveMove.eOpClCtrl := E_OpClCtrl.Close;
		nStateA_OpenClose := 60;
		nStateA_OpenCloseNext := 2;
		
	2:	//vertikal öffnen
		eReactDrive := E_ReactDrive.CoverVerti;
		fbReactDriveMove.eOpClCtrl := E_OpClCtrl.Open;
		nStateA_OpenClose := 60;
		nStateA_OpenCloseNext := 3;
	
	3:	//horizontal öffnen
		eReactDrive := E_ReactDrive.CoverHoriz;
		nStateA_OpenClose := 60;
		nStateA_OpenCloseNext := 4;
		
	4:	//Clamp öffnen
		eReactDrive := E_ReactDrive.Clamp;
		nStateA_OpenClose := 60;
		nStateA_OpenCloseNext := 80;
	
		////////////////////////////////CoverBoth close//////////////////////////////////////////////
	5:	//horizontal schließen
		eReactDrive := E_ReactDrive.CoverHoriz;
		nStateA_OpenClose := 60;
		nStateA_OpenCloseNext := 6;

	6:	//vertikal schließen 
		eReactDrive := E_ReactDrive.CoverVerti;
		nStateA_OpenClose := 60;
		nStateA_OpenCloseNext := 80;
		
		////////////////////////////////Complete öffnen////////////////////////////////////////////
	10:	//vertikal öffnen
		eReactDrive := E_ReactDrive.CoverVerti;
		nStateA_OpenClose := 60;
		nStateA_OpenCloseNext := 11;
		
	11:	//horizontal öffnen
		eReactDrive := E_ReactDrive.CoverHoriz;
		nStateA_OpenClose := 60;
		nStateA_OpenCloseNext := 12;
	
	12:	//Clamp öffen
		eReactDrive := E_ReactDrive.Clamp;
		nStateA_OpenClose := 60;
		nStateA_OpenCloseNext := 80;
		
		////////////////////////////////Complete schließen////////////////////////////////////////////
	13: //Clamp schließen
		eReactDrive := E_ReactDrive.Clamp;
		nStateA_OpenClose := 60;
		nStateA_OpenCloseNext := 14;
		
	14:	//horizontal schließen
		eReactDrive := E_ReactDrive.CoverHoriz;
		nStateA_OpenClose := 60;
		nStateA_OpenCloseNext := 15;
	
	15:	//vertikal schließen
		eReactDrive := E_ReactDrive.CoverVerti;
		nStateA_OpenClose := 60;
		nStateA_OpenCloseNext := 80;
END_CASE

IF nStateA_OpenClose = 60 THEN
	fbReactDriveMove(pDriveRef:= pDriveRef, eDrive:= eReactDrive, bExecute:= TRUE);
	IF NOT fbReactDriveMove.bBusy THEN
		IF fbReactDriveMove.bError THEN
			stError.ErrorId := fbReactDriveMove.nErrorId;
			nStateA_OpenClose := 99;
		ELSE
			nStateA_OpenClose := nStateA_OpenCloseNext;
		END_IF
		fbReactDriveMove(bExecute:= FALSE);
	END_IF	
ELSIF nStateA_OpenClose = 70 THEN
	//Abbrechen
	;
END_IF

//Errorhandling
IF nStateA_OpenClose = 99 THEN
	stError.Cmd := E_Action.ACTION_ReactorOpCl;
	stError.POUAction := E_POUACT.POUACT_A_OpenClose;
	fbErrorList.M_Add(stError);
END_IF
END_ACTION

ACTION A_Reset:
CASE nStateA_Reset OF
	0:
		nStateA_Reset := 80;
END_CASE
END_ACTION

ACTION A_Stop:
CASE nStateA_Stop OF
	0:
		IF nStateA_Init < 70 AND bInit THEN	//Initialisieren abbrechen
			nStateA_Init := 70;
		END_IF
		
		IF bCooling AND nStateA_Cooling < 70 THEN
			nStateA_Cooling := 70;
		END_IF
		
		nStateA_Stop := 1;
		
	1:	//Warten bis alle Actions fertig abgebrochen
		IF hList.nCount = 1 THEN	//nur der Eintrag von Stop
			nStateA_Stop := 80;
		END_IF

END_CASE
END_ACTION

METHOD FB_init : BOOL
VAR_INPUT
	bInitRetains : BOOL; // if TRUE, the retain variables are initialized (warm start / cold start)
	bInCopyCode : BOOL;  // if TRUE, the instance afterwards gets moved into the copy code (online change)
END_VAR
eObjectType := E_ObjectType.OBJECTTYPE_Reactor;
eObjectGroup := E_ObjectGroup.OBJECTGROUP_Target OR E_ObjectGroup.OBJECTGROUP_Device;
END_METHOD

METHOD M_AddChild : ERRORID
VAR_INPUT
	pObject : POINTER TO FB_Object;
	nSlotNr	: UINT;
	nIndex 	: INT;	
END_VAR
IF pObject > 0 THEN
	IF nSlotNr = fbVialSlot.P_nNr THEN //Reactor besitzt nur den VialSlot
		IF fbVialSlot.P_pChild = 0 THEN
			//Object darf selber noch an keinem Parent hängen
			IF pObject^.P_pParentObject = 0 THEN
				fbVialSlot.P_pChild := pObject;
				pObject^.P_pObjCollectNode := pObjCollectNode^.nodes.M_AddNewNode(pObject,nIndex);
				pObject^.M_UpdateParent();
			ELSE
				M_AddChild := E_ErrorIdObjMgmt.ERRORID_ObjectAlreadyOnAnotherParent;
			END_IF
		ELSE //Slot bereits belegt
			M_AddChild := E_ErrorIdObjMgmt.ERRORID_SlotIsAlreadyOccupied;
		END_IF		
	ELSE
		M_AddChild := SUPER^.M_AddChild(pObject,nSlotNr,nIndex);
	END_IF
ELSE
	M_AddChild := E_ErrorIdObjMgmt.ERRORID_InvalidParentObject;
END_IF
END_METHOD

METHOD M_ApplyPos : ERRORID
VAR_INPUT
	eTargetRef 		: E_TargetRef;
	nPointSlotNr	: UINT;
	stPos 			: ST_3DPoint;
	bXPos			: BOOL;
	bYPos			: BOOL;
	bZPos			: BOOL;	
END_VAR

VAR
	stAbsPos		: ST_3DPoint;
END_VAR
IF eTargetRef = E_TargetRef.TARGETREF_Slot THEN
	IF nPointSlotNr = 1 THEN
		stAbsPos := P_stAbsPosLB;
		IF bXPos THEN
			fbVialSlot.P_rRelPosX := stPos.X - stAbsPos.X;	
		END_IF
		IF bYPos THEN
			fbVialSlot.P_rRelPosY := stPos.Y - stAbsPos.Y;	
		END_IF
		IF bZPos THEN
			fbVialSlot.P_rRelPosZ := stPos.Z - stAbsPos.Z;	
		END_IF
	ELSE
		M_ApplyPos := E_ErrorIdCmd.ERRORID_InvalidTargetPointNr;
	END_IF
ELSE
	M_ApplyPos := SUPER^.M_ApplyPos(eTargetRef, nPointSlotNr, stPos,bXPos,bYPos,bZPos);
END_IF
END_METHOD

METHOD M_CancelAction
VAR_INPUT
	eAction : E_Action;
END_VAR
IF eAction = E_Action.ACTION_Cooling THEN
	IF bCooling AND nStateA_Cooling < 70 THEN
		nStateA_Cooling := 70;
	END_IF
END_IF
END_METHOD

METHOD M_CheckAction : ERRORID
VAR_INPUT
	refActionData 	: REFERENCE TO ST_ActionData;
	pCorrelObject	: POINTER TO FB_Object;
END_VAR

VAR
	pPiece : POINTER TO FB_PieceBase;
	pVial : POINTER TO FB_Vial;
END_VAR
IF refActionData.eAction = E_Action.ACTION_TeachTarget THEN
	IF NOT DINT_TO_UINT(refActionData.aParams[1]) = E_TargetRef.TARGETREF_SpecPoint AND refActionData.aParams[2] = 1 THEN
		M_CheckAction := E_ErrorIdCmd.ERRORID_InvalidTargetPointRef;
	END_IF
ELSIF refActionData.eAction = E_Action.ACTION_ExchangePiece THEN
	//Slot gültig?
	IF refActionData.aParams[1] <> 1 THEN
		M_CheckAction := E_ErrorIdCmd.ERRORID_InvalidTargetSlot;
		RETURN;
	END_IF
	pPiece := pCorrelObject;
	IF refActionData.aParams[2] = 0 THEN //Drop
		//Hier wird das zu handlende Piece benötigt
		IF pPiece^.P_eObjectType = E_ObjectType.OBJECTTYPE_Septum THEN
			//Es muss Vial in Slot sein
			IF fbVialSlot.P_pPiece = 0 THEN
				M_CheckAction := E_ErrorIdCmd.ERRORID_NoPieceInSlot;
				RETURN;				
			END_IF
			//Es darf noch kein Septum am Vial sein
			pVial := fbVialSlot.P_pPiece;
			IF pVial^.P_pSeptum > 0 THEN
				M_CheckAction := E_ErrorIdCmd.ERRORID_SeptumAlreadyOnVial;
			END_IF
		ELSIF pPiece^.P_eObjectType = E_ObjectType.OBJECTTYPE_Vial THEN
			//Es darf noch kein Vial im Slot sein
			IF fbVialSlot.P_pPiece > 0 THEN
				M_CheckAction := E_ErrorIdCmd.ERRORID_PieceAlreadyInSlot;
			END_IF
		ELSE
			M_CheckAction := E_ErrorIdCmd.ERRORID_InvalidPieceType;
		END_IF
	END_IF
ELSIF refActionData.eAction = E_Action.ACTION_DockTool THEN
	//Im Slot muss ein Vial sein, welches aber kein Septum hat
	//Der Reaktor muss offen sein
	pVial := fbVialSlot.P_pPiece;
	IF pVial > 0 THEN
		IF pVial^.P_pSeptum > 0 THEN //Error
			M_CheckAction := E_ErrorIdCmd.ERRORID_SeptumAlreadyOnVial;
		ELSE
			IF pDriveRef^.eCurrentState[E_ReactDrive.CoverHoriz] <> E_OpClState.Open THEN
				M_CheckAction := E_ErrorIdCmd.ERRORID_ReactorNotOpen;
			END_IF
 		END_IF
	ELSE //Error
		M_CheckAction := E_ErrorIdCmd.ERRORID_NoPieceInSlot;
	END_IF
ELSIF refActionData.eAction = E_Action.ACTION_InsertTool THEN
	//Im Slot muss ein Vial sein, welches aber kein Septum hat
	//Der Reaktor muss offen sein
	pVial := fbVialSlot.P_pPiece;
	IF pVial > 0 THEN
		IF pVial^.P_pSeptum > 0 THEN //Error
			M_CheckAction := E_ErrorIdCmd.ERRORID_SeptumAlreadyOnVial;
		ELSE
			IF pDriveRef^.eCurrentState[E_ReactDrive.CoverHoriz] <> E_OpClState.Open THEN
				M_CheckAction := E_ErrorIdCmd.ERRORID_ReactorNotOpen;
			END_IF
 		END_IF
	ELSE //Error
		M_CheckAction := E_ErrorIdCmd.ERRORID_NoPieceInSlot;
	END_IF
ELSIF refActionData.eAction = E_Action.ACTION_MoveToTarget THEN
	//Falls zu Slot gefahren werden soll, dann muss Reactor offen sein
	IF refActionData.aParams[1] = E_TargetRef.TARGETREF_Slot THEN
		IF pDriveRef^.eCurrentState[E_ReactDrive.CoverHoriz] <> E_OpClState.Open THEN
			M_CheckAction := E_ErrorIdCmd.ERRORID_ReactorNotOpen;
		END_IF
	END_IF
ELSE
	M_CheckAction := E_ErrorIdCmd.ERRORID_InvalidAction;
END_IF
END_METHOD

METHOD M_CheckProcDataType : BOOL
VAR_INPUT
	eProcDataType : E_ProcDataType;
END_VAR
IF eProcDataType = E_ProcDataType.PROCDATATYPE_Temp1 THEN
	M_CheckProcDataType := TRUE;
END_IF
END_METHOD

METHOD M_ClearAllProps
VAR_INPUT
	bIgnoreParent : BOOL; //Es wird das gesamte OD gelöscht. -> Zeiger auf Parent nicht mehr gültig!
END_VAR
SUPER^.M_ClearAllProps(bIgnoreParent);
fbVialSlot.P_pPiece := 0;
END_METHOD

METHOD M_ExeAction : ERRORID
VAR_INPUT
	refActionData	: REFERENCE TO ST_ActionData;
END_VAR
IF NOT (eCurrentState = E_MachineState.MACHINESTATE_Idle OR
	eCurrentState = E_MachineState.MACHINESTATE_Active OR
	eCurrentState = E_MachineState.MACHINESTATE_Ready) THEN
	M_ExeAction := E_ErrorIdCmd.ERRORID_InvalidState;
	RETURN;
END_IF

CASE refActionData.eAction OF
	E_Action.ACTION_Init:
		IF NOT bInit THEN
			bInit := TRUE;
			fbList.A_AddHeadValue(hList := hList, putValue:= E_Action.ACTION_Init);
			bIsInit := FALSE;
		ELSE
			RETURN;
		END_IF
		
	E_Action.ACTION_Heating:	//Heizung ON/OFF
			IF pHeaterRef = 0 THEN
				M_ExeAction := E_ErrorIdObjMgmt.ERRORID_InvalidHardwareRef;
				RETURN;
			END_IF
			nTempSetpoint := DINT_TO_USINT(refActionData.aParams[1]/10);
			bHeaterOn := DINT_TO_BOOL(refActionData.aParams[2]);
			IF bHeaterOn THEN
				IF nTempSetpoint > 100 THEN
					M_ExeAction := E_ErrorIdCmd.ERRORID_InvalidHeatingTemp;
					RETURN;
				END_IF
			IF bCooling THEN
				nStateA_Cooling := 70;
			END_IF				
			END_IF
			pHeaterRef^.P_nTempSetpoint := nTempSetpoint;
			pHeaterRef^.P_bHeatingOn := bHeaterOn;
			
	E_Action.ACTION_Cooling:	//Kühlung ON/OFF
		nTempCooling := DINT_TO_UINT(refActionData.aParams[1]);
		bCoolingOn := DINT_TO_BOOL(refActionData.aParams[2]);
		IF bCoolingOn AND NOT bCooling THEN
 			bCooling := TRUE;
			fbList.A_AddHeadValue(hList := hList, putValue:= E_Action.ACTION_Cooling);
		ELSE
			IF bCooling THEN
				nStateA_Cooling := 70;
			END_IF
		END_IF
		
	E_Action.ACTION_DetectVial:
		IF pHeaterRef = 0 THEN
			M_ExeAction := E_ErrorIdObjMgmt.ERRORID_InvalidHardwareRef;
			RETURN;
		END_IF
	
		IF NOT bDetectVial THEN
			eEndState := DINT_TO_USINT(refActionData.aParams[1]);
			fbList.A_AddHeadValue(hList := hList, putValue:= E_Action.ACTION_DetectVial);
			bDetectVial := TRUE;						
		ELSE
			M_ExeAction := E_ErrorIdCmd.ERRORID_BasicActionActive;
			RETURN;
		END_IF
	
	E_Action.ACTION_ReactorOpCl:
		IF NOT bOpenClose THEN
			eReactComponent := DINT_TO_USINT(refActionData.aParams[1]);
			eOpClCtrl := DINT_TO_USINT(refActionData.aParams[2]);
			IF eReactComponent = E_ReactDrive.CoverHoriz OR  eReactComponent = E_ReactDrive.CoverBoth OR 
				eReactComponent = E_ReactDrive.Complete THEN
				IF eOpClCtrl = E_OpClCtrl.Close THEN
					IF NOT P_bCoverAreaIsFree THEN
						M_ExeAction := E_ErrorIdCmd.ERRORID_ReactorCoverNotFree;
						RETURN;			
					END_IF
				END_IF
			END_IF
			fbList.A_AddHeadValue(hList := hList, putValue:= E_Action.ACTION_ReactorOpCl);
			bOpenClose := TRUE;
		ELSE
			M_ExeAction := E_ErrorIdCmd.ERRORID_BasicActionActive;
			RETURN;
		END_IF
		
	E_Action.ACTION_Stop:
		//Stop braucht nur ausgeführt werden, wenn irgendwas aktiv ist
		IF bBusy AND nStateA_Stop = 0 AND hList.nCount > 0 THEN
			bStop := TRUE;
			fbList.A_AddHeadValue(hList := hList, putValue := E_Action.ACTION_Stop);
		ELSE
			RETURN;
		END_IF
	ELSE
		M_ExeAction := E_ErrorIdCmd.ERRORID_InvalidAction;
END_CASE

bBusy := TRUE;
eCurrentState := E_MachineState.MACHINESTATE_Active;
END_METHOD

METHOD M_GetAbsPos : ST_3DPoint
VAR_INPUT
	pChildPos	: POINTER TO ST_3DPoint;
	eTargetRef 	: E_TargetRef;
	nParam1		: UINT;
 	nParam2		: UINT;
	nParam3		: USINT;
	nParam4		: USINT;
	nZLevel		: USINT;
END_VAR
VAR_OUTPUT
	nErrorId 	: ERRORID;
	lrAngle		: LREAL;
END_VAR
VAR
	stLocPosLB : ST_3DPoint;
END_VAR
IF eTargetRef = E_TargetRef.TARGETREF_Slot THEN
	IF nParam1 = 1 THEN
		stLocPosLB := P_stRelPosLB;
		//Slot belegt?
		IF fbVialSlot.P_pPiece > 0 THEN
			stLocPosLB := F_Add3DPoints(stLocPosLB, fbVialSlot.P_pPiece^.M_GetRelPosTopCenter());
		ELSE
			stLocPosLB := F_Add3DPoints(stLocPosLB,fbVialSlot.P_stRelPos);	
		END_IF
		
		M_GetAbsPos := pParentTarget^.M_GetAbsPos(pChildPos := ADR(stLocPosLB), eTargetRef:= E_TargetRef.TARGETREF_LeftBottom,
													nParam1:= 0,
													nParam2:= 0, nParam3:= 0, nParam4:= 0, nZLevel:= 0,
													lrAngle => lrAngle, nErrorId=> nErrorId);		
	ELSE
		nErrorId := E_ErrorIdCmd.ERRORID_InvalidTargetPointNr;
	END_IF
ELSE
	M_GetAbsPos := SUPER^.M_GetAbsPos(pChildPos := pChildPos, eTargetRef:= eTargetRef,
													nParam1:= nParam1,
													nParam2:= nParam2, nParam3:= nParam3, nParam4:= 0, nZLevel:= nZLevel,
													lrAngle => lrAngle, nErrorId=> nErrorId);		
END_IF
END_METHOD

METHOD M_GetActionBusy : BOOL
VAR_INPUT
	eAction : E_Action;
END_VAR
getPosPtr := 0;(* start from first node element *)
fbList.A_FindNext( hList := hList, putPosPtr := getPosPtr, putValue := eAction, getValue=>getValue, getPosPtr=>getPosPtr );
IF fbList.bOk THEN	//Eintrag wurde gefunden, d.h. Action ist noch busy
	M_GetActionBusy := TRUE;
END_IF
END_METHOD

METHOD M_GetAllProps : ERRORID
VAR_INPUT
	refCmdData : REFERENCE TO  ST_CmdData;
END_VAR

VAR
END_VAR
SUPER^.M_GetAllProps(refCmdData);
nCurrentPropIndex := nCurrentPropIndex + 1;
refCmdData.n32Data[nCurrentPropIndex] := nNoOfSlots;
nCurrentPropIndex := nCurrentPropIndex + 1;
refCmdData.n32Data[nCurrentPropIndex] := fbVialSlot.nNr;
nCurrentPropIndex := nCurrentPropIndex + 1;
refCmdData.n32Data[nCurrentPropIndex] := REAL_TO_DINT(fbVialSlot.P_rRelPosX);
nCurrentPropIndex := nCurrentPropIndex + 1;
refCmdData.n32Data[nCurrentPropIndex] := REAL_TO_DINT(fbVialSlot.P_rRelPosY);
nCurrentPropIndex := nCurrentPropIndex + 1;
refCmdData.n32Data[nCurrentPropIndex] := REAL_TO_DINT(fbVialSlot.P_rRelPosZ);
nCurrentPropIndex := nCurrentPropIndex + 1;
refCmdData.n32Data[nCurrentPropIndex] := REAL_TO_DINT(fbVialSlot.P_rDepth);

//ReglerParamter der Heaters
IF pHeaterRef > 0 THEN
	nCurrentPropIndex := nCurrentPropIndex + 1;
	refCmdData.n32Data[nCurrentPropIndex] := pHeaterRef^.P_nPidKp;
	nCurrentPropIndex := nCurrentPropIndex + 1;
	refCmdData.n32Data[nCurrentPropIndex] := pHeaterRef^.P_nPidKi;
	nCurrentPropIndex := nCurrentPropIndex + 1;
	refCmdData.n32Data[nCurrentPropIndex] := pHeaterRef^.P_nPidKd;
	nCurrentPropIndex := nCurrentPropIndex + 1;
	refCmdData.n32Data[nCurrentPropIndex] := pHeaterRef^.P_nPidTa;
ELSE
	nCurrentPropIndex := nCurrentPropIndex + 4;
END_IF

nCurrentPropIndex := nCurrentPropIndex + 1;
refCmdData.n32Data[nCurrentPropIndex] := nValveNrCool;

//ClosedPositionen
nCurrentPropIndex := nCurrentPropIndex + 1;
refCmdData.n32Data[nCurrentPropIndex] := pDriveRef^.nClosedPosition[1];
nCurrentPropIndex := nCurrentPropIndex + 1;
refCmdData.n32Data[nCurrentPropIndex] := pDriveRef^.nClosedPosition[2];
nCurrentPropIndex := nCurrentPropIndex + 1;
refCmdData.n32Data[nCurrentPropIndex] := pDriveRef^.nClosedPosition[3];

//MoveSpeeds
nCurrentPropIndex := nCurrentPropIndex + 1;
refCmdData.n32Data[nCurrentPropIndex] := pDriveRef^.nMotorSpeed[1];
nCurrentPropIndex := nCurrentPropIndex + 1;
refCmdData.n32Data[nCurrentPropIndex] := pDriveRef^.nMotorSpeed[2];
nCurrentPropIndex := nCurrentPropIndex + 1;
refCmdData.n32Data[nCurrentPropIndex] := pDriveRef^.nMotorSpeed[3];
END_METHOD

METHOD M_GetProcData : DINT
VAR_INPUT
	eProcDataType : E_ProcDataType;
END_VAR
IF eProcDataType = E_ProcDataType.PROCDATATYPE_Temp1 THEN
	M_GetProcData := nTempActual;
END_IF
END_METHOD

METHOD M_GetSlot : POINTER TO FB_Slot
VAR_INPUT
	nSlotNr : UINT;
END_VAR
IF nSlotNr = 1 THEN
	M_GetSlot := ADR(fbVialSlot);
END_IF
END_METHOD

METHOD M_GetSlotFromChild : POINTER TO FB_Slot
VAR_INPUT
	pObject : POINTER TO FB_Object;
END_VAR
IF fbVialSlot.P_pChild = pObject THEN
	M_GetSlotFromChild := ADR(fbVialSlot);
END_IF
END_METHOD

METHOD M_RemoveListEntry : BOOL
VAR_INPUT
	nSearchValue : E_Action;
END_VAR
getPosPtr := 0;(* start from first node element *)
fbList.A_FindNext( hList := hList, putPosPtr := getPosPtr, putValue := nSearchValue, getValue=>getValue, getPosPtr=>getPosPtr );
IF fbList.bOk THEN	//Eintrag wurde gefunden
	fbList.A_RemoveValueAtPosPtr(hList:= hList,	putPosPtr:= getPosPtr);
	IF fbList.bOk THEN
		M_RemoveListEntry := TRUE;
	END_IF
END_IF
END_METHOD

METHOD M_SetAllProps : ERRORID
VAR_INPUT
	refCmdData : REFERENCE TO  ST_CmdData;
END_VAR

VAR
END_VAR
{IF defined (variable:aFbReactDriveRef)}
pDriveRef := ADR(aFbReactDriveRef[1]);
{ELSE}
M_SetAllProps := E_ErrorIdObjMgmt.ERRORID_InvalidHardwareRef;
{END_IF}

M_SetAllProps := SUPER^.M_SetAllProps(refCmdData);

IF M_SetAllProps > 0 THEN
	RETURN;
END_IF

nCurrentPropIndex := nCurrentPropIndex + 1;
nSpecPropIndex := nCurrentPropIndex;
//NumberOfSlots immer "1"
nNoOfSlots := DINT_TO_USINT(refCmdData.n32Data[nCurrentPropIndex]);
IF nNoOfSlots <> 1 THEN
	nNoOfSlots := 1;
	M_SetAllProps := E_ErrorIdObjMgmt.ERRORID_InvalidNoOfSlots;
	RETURN;
END_IF
nCurrentPropIndex := nCurrentPropIndex + 1;
fbVialSlot.P_nNr := DINT_TO_UINT(refCmdData.n32Data[nCurrentPropIndex]);
//SlotNr immer "1"
IF fbVialSlot.P_nNr <> 1 THEN
	fbVialSlot.P_nNr := 1;
	M_SetAllProps := E_ErrorIdObjMgmt.ERRORID_InvalidSlotNumber;
	RETURN;
END_IF

nCurrentPropIndex := nCurrentPropIndex + 1;
fbVialSlot.P_rRelPosX := DINT_TO_REAL(refCmdData.n32Data[nCurrentPropIndex]);
nCurrentPropIndex := nCurrentPropIndex + 1;
fbVialSlot.P_rRelPosY := DINT_TO_REAL(refCmdData.n32Data[nCurrentPropIndex]);
nCurrentPropIndex := nCurrentPropIndex + 1;
fbVialSlot.P_rRelPosZ := DINT_TO_REAL(refCmdData.n32Data[nCurrentPropIndex]);
nCurrentPropIndex := nCurrentPropIndex + 1;
fbVialSlot.P_rDepth := DINT_TO_REAL(refCmdData.n32Data[nCurrentPropIndex]);

{IF defined (variable:aFbReactHeatRef)}
pHeaterRef := ADR(aFbReactHeatRef[1]);
nCurrentPropIndex := nCurrentPropIndex + 1;
pHeaterRef^.P_nPidKp := DINT_TO_UINT(refCmdData.n32Data[nCurrentPropIndex]);
nCurrentPropIndex := nCurrentPropIndex + 1; 
pHeaterRef^.P_nPidKi := DINT_TO_UINT(refCmdData.n32Data[nCurrentPropIndex]);
nCurrentPropIndex := nCurrentPropIndex + 1;
pHeaterRef^.P_nPidKd := DINT_TO_UINT(refCmdData.n32Data[nCurrentPropIndex]);
nCurrentPropIndex := nCurrentPropIndex + 1;
pHeaterRef^.P_nPidTa := DINT_TO_USINT(refCmdData.n32Data[nCurrentPropIndex]);
{ELSE}
{warning 'implement errorId}
M_SetAllProps := 5555;
{END_IF}
{IF defined (variable:aFbReactHeatRef)}


{END_IF}
nCurrentPropIndex := nCurrentPropIndex + 1;
IF refCmdData.n32Data[nCurrentPropIndex] > 0 AND refCmdData.n32Data[nCurrentPropIndex] <= cNoOfValves THEN
	nValveNrCool := DINT_TO_USINT(refCmdData.n32Data[nCurrentPropIndex]);
ELSE
	M_SetAllProps := E_ErrorIdObjMgmt.ERRORID_InvalidValveNumber;
END_IF

//ClosedPositionen
nCurrentPropIndex := nCurrentPropIndex + 1;
pDriveRef^.nClosedPosition[1] := refCmdData.n32Data[nCurrentPropIndex];
nCurrentPropIndex := nCurrentPropIndex + 1;
pDriveRef^.nClosedPosition[2] := refCmdData.n32Data[nCurrentPropIndex];
nCurrentPropIndex := nCurrentPropIndex + 1;
pDriveRef^.nClosedPosition[3] := refCmdData.n32Data[nCurrentPropIndex];
//MoveSpeeds
nCurrentPropIndex := nCurrentPropIndex + 1;
pDriveRef^.nMotorSpeed[1] := refCmdData.n32Data[nCurrentPropIndex];
nCurrentPropIndex := nCurrentPropIndex + 1;
pDriveRef^.nMotorSpeed[2] := refCmdData.n32Data[nCurrentPropIndex];
nCurrentPropIndex := nCurrentPropIndex + 1;
pDriveRef^.nMotorSpeed[3] := refCmdData.n32Data[nCurrentPropIndex];

nNoOfProps := nCurrentPropIndex + 1;
END_METHOD

METHOD M_SetSingleProp : ERRORID
VAR_INPUT
	refCmdData : REFERENCE TO  ST_CmdData;
END_VAR
IF nSpecPropIndex = refCmdData.aHeader[1] THEN //Anzahl Slots darf nicht verändert werden
	M_SetSingleProp := E_ErrorIdCmd.ERRORID_InvalidProperty;
ELSIF (nSpecPropIndex + 1) = refCmdData.aHeader[1] THEN
	M_SetSingleProp := E_ErrorIdCmd.ERRORID_InvalidProperty; //SlotNr darf nicht verändert werden
ELSIF (nSpecPropIndex + 2) = refCmdData.aHeader[1] THEN
	fbVialSlot.P_rRelPosX := DINT_TO_REAL(refCmdData.n32Data[0]);
ELSIF (nSpecPropIndex + 3) = refCmdData.aHeader[1] THEN
	fbVialSlot.P_rRelPosY := DINT_TO_REAL(refCmdData.n32Data[0]);
ELSIF (nSpecPropIndex + 4) = refCmdData.aHeader[1] THEN
	fbVialSlot.P_rRelPosZ := DINT_TO_REAL(refCmdData.n32Data[0]);
ELSIF (nSpecPropIndex + 5) = refCmdData.aHeader[1] THEN
	fbVialSlot.P_rDepth := DINT_TO_REAL(refCmdData.n32Data[0]);
ELSIF (nSpecPropIndex + 6) = refCmdData.aHeader[1] THEN
	IF pHeaterRef > 0 THEN
		pHeaterRef^.P_nPidKp := DINT_TO_UINT(refCmdData.n32Data[0]);
	ELSE
		M_SetSingleProp := E_ErrorIdCmd.ERRORID_InvalidProperty;
	END_IF	
ELSIF (nSpecPropIndex + 7) = refCmdData.aHeader[1] THEN
	IF pHeaterRef > 0 THEN
		pHeaterRef^.P_nPidKi := DINT_TO_UINT(refCmdData.n32Data[0]);
	ELSE
		M_SetSingleProp := E_ErrorIdCmd.ERRORID_InvalidProperty;
	END_IF	
ELSIF (nSpecPropIndex + 8) = refCmdData.aHeader[1] THEN
	IF pHeaterRef > 0 THEN
		pHeaterRef^.P_nPidKd := DINT_TO_UINT(refCmdData.n32Data[0]);
	ELSE
		M_SetSingleProp := E_ErrorIdCmd.ERRORID_InvalidProperty;
	END_IF	
ELSIF (nSpecPropIndex + 9) = refCmdData.aHeader[1] THEN
	IF pHeaterRef > 0 THEN
		pHeaterRef^.P_nPidTa := DINT_TO_USINT(refCmdData.n32Data[0]);
	ELSE
		M_SetSingleProp := E_ErrorIdCmd.ERRORID_InvalidProperty;
	END_IF	
ELSIF (nSpecPropIndex + 10) = refCmdData.aHeader[1] THEN
	IF refCmdData.n32Data[0] > 0 AND refCmdData.n32Data[0] <= cNoOfValves THEN
		nValveNrCool := DINT_TO_USINT(refCmdData.n32Data[0]);
	ELSE
		M_SetSingleProp := E_ErrorIdObjMgmt.ERRORID_InvalidValveNumber;
	END_IF
ELSIF (nSpecPropIndex + 11) = refCmdData.aHeader[1] THEN
	pDriveRef^.nClosedPosition[1] := refCmdData.n32Data[0];
ELSIF (nSpecPropIndex + 12) = refCmdData.aHeader[1] THEN
	pDriveRef^.nClosedPosition[2] := refCmdData.n32Data[0];
ELSIF (nSpecPropIndex + 13) = refCmdData.aHeader[1] THEN
	pDriveRef^.nClosedPosition[3] := refCmdData.n32Data[0];
ELSIF (nSpecPropIndex + 14) = refCmdData.aHeader[1] THEN
	pDriveRef^.nMotorSpeed[1] := refCmdData.n32Data[0];
ELSIF (nSpecPropIndex + 15) = refCmdData.aHeader[1] THEN
	pDriveRef^.nMotorSpeed[2] := refCmdData.n32Data[0];
ELSIF (nSpecPropIndex + 16) = refCmdData.aHeader[1] THEN
	pDriveRef^.nMotorSpeed[3] := refCmdData.n32Data[0];
ELSE
	M_SetSingleProp := SUPER^.M_SetSingleProp(refCmdData);
END_IF
END_METHOD

METHOD PRIVATE M_SetSpeed : BOOL
VAR_INPUT
	nSpeed : UDINT;
END_VAR

VAR_OUTPUT
	nErrorId	: ERRORID;
END_VAR
(*//Profile Speed setzen
fbSdoWrite(sADSNetID:= stPowdStatRef.stAdsAdress.sNetId,nPortNr:= stPowdStatRef.stAdsAdress.nPort, 
			nIndex:= 16#6081, nSubIndex:= 0, nDataLength:= 4, nData:= UDINT_TO_DINT(nSpeed), bExecute:= TRUE);

M_SetSpeed := fbSdoWrite.bBusy; 

IF NOT fbSdoWrite.bBusy THEN
	IF fbSdoWrite.bError THEN
		nErrorId := fbSdoWrite.nAdsErrorId;
	END_IF
	fbSdoWrite(bExecute:= FALSE);
END_IF			
*)
END_METHOD

METHOD M_Stop : ERRORID
VAR_INPUT
END_VAR
//Stop braucht nur ausgeführt werden, wenn irgendwas aktiv ist
IF NOT bStop AND eCurrentState = E_MachineState.MACHINESTATE_Active THEN
 	//stPowdStatRef.bShaker := FALSE;
	bStop := TRUE;
	fbList.A_AddHeadValue(hList := hList, putValue := E_Action.ACTION_Stop);
END_IF
END_METHOD

METHOD M_TakePiece : POINTER TO FB_PieceSlot
VAR_INPUT
	pPiece : POINTER TO FB_PieceBase;
	nSlotNr : UINT;
END_VAR
IF pPiece > 0 THEN
	IF 	nSlotNr = 1 THEN
		//Slot frei?
		IF fbVialSlot.P_pPiece = 0 THEN
			fbVialSlot.P_pPiece := pPiece;
			M_TakePiece := ADR(fbVialSlot);
		END_IF
	END_IF
END_IF
END_METHOD

PROPERTY P_bCoverAreaIsFree : BOOL
GET
VAR
	i : UINT;
	stCurPosMzTool	: ST_3DPoint;
	stCurPosThis	: ST_3DPoint;
END_VAR
//Checken, ob sich im Bewegungsbereich des Deckel ein MzTool befindet
P_bCoverAreaIsFree := TRUE;
(*FOR i:= 1 TO fbObjectDirectory.nCntMzTool BY 1 DO
	IF NOT (aI_MzTool[i].P_eObjectType = E_ObjectType.OBJECTTYPE_MZHead) THEN
		IF NOT aI_MzTool[i].P_bCollFree THEN	//Tool ist nicht im kollisionsfreiem Bereich
			
			stCurPosMzTool := aI_MzTool[i].P_stCurrentPosPhys;
			stCurPosThis := P_stAbsPosLB;
			IF (stCurPosMzTool.Z - 2000) < stCurPosThis.Z THEN //MzTool befindet sich 5mm unterhalb der Oberkante Reaktor und in dessen XY Bereich
				IF stCurPosMzTool.X >= stCurPosThis.X AND stCurPosMzTool.X <= (stCurPosThis.X + stDimension.Width)
				AND stCurPosMzTool.Y >= stCurPosThis.Y AND stCurPosMzTool.Y <= (stCurPosThis.Y + stDimension.Depth) THEN
					P_bCoverAreaIsFree := FALSE;
					RETURN;
				END_IF
			END_IF
 		END_IF
	END_IF
END_FOR*)
END_GET
END_PROPERTY

PROPERTY P_bVialInSlot : BOOL
GET
IF pHeaterRef > 0 THEN
	P_bVialInSlot := pHeaterRef^.P_bVialDetected;
END_IF
END_GET
END_PROPERTY

PROPERTY P_pVial : POINTER TO FB_Vial
GET
P_pVial := fbVialSlot.P_pPiece;
END_GET
SET
fbVialSlot.P_pPiece := P_pVial;
END_SET
END_PROPERTY

END_FUNCTION_BLOCK

// ---- Hardware/Reactor/FB_HwRefReactDrive.TcPOU
FUNCTION_BLOCK FB_HwRefReactDrive EXTENDS FB_CanNodeBase
VAR_INPUT
	//Ausgänge
	nControl	AT %Q* : ARRAY[1..3] OF UINT;	//Controlword
	nOpMode		AT %Q* : ARRAY[1..3] OF USINT;	//Mode of Operation
	nTargetPos	AT %Q* : ARRAY[1..3] OF DINT;	//TargetPos
	nClosedPosition : ARRAY[1..3] OF DINT;
	nMotorSpeed : ARRAY[1..3] OF DINT;
	eCurrentState : ARRAY[1..3] OF E_OpClState;
	bIsInit : BOOL;
END_VAR
VAR_OUTPUT
	//Eingänge
	nStatus			AT %I* : ARRAY[1..3] OF UINT;	//Statusword
	nCurrentOpMode	AT %I* : ARRAY[1..3] OF USINT; //Aktueller Wert von Mode of Operation
END_VAR
VAR
	
END_VAR

IF bNodeEnabled THEN
	SUPER^();	
END_IF

END_FUNCTION_BLOCK

// ---- Hardware/Reactor/FB_HwRefReactHeater.TcPOU
FUNCTION_BLOCK FB_HwRefReactHeater EXTENDS FB_CanNodeBase
VAR_INPUT
END_VAR
VAR_OUTPUT
END_VAR
VAR
	//Eingänge
	nTempActual 	AT %I* : UINT;	//aktuelle Temperatur in 1/100tel °C 
	bTempCutoff 	AT %I* : BOOL;	//Übertemperaturabschaltung wurde aktiviert
	bVialDetected	AT %I* : BOOL;
	//Ausgänge
	nPidKp 			AT %Q* : UINT; 	//PID-Reglerparameter KP
	nPidKi 			AT %Q* : UINT;	//PID-Reglerparameter KI
	nPidKd 			AT %Q* : UINT;	//PID-Reglerparameter KD
	nPidTa 			AT %Q* : USINT;	//PID-Reglerparameter TA
	bHeatingOn		AT %Q* : BOOL;	//Heizer EIN
	nTempSetpoint	AT %Q* : USINT;	//Solltemperatur in °C (ohne Kommastellen)
	bResetVialDetect AT %Q* : BOOL;	//VialDetection zurücksetzen
END_VAR

IF bNodeEnabled THEN
	SUPER^();
END_IF

PROPERTY P_bHeatingOn : BOOL
SET
bHeatingOn := P_bHeatingOn;
END_SET
GET
P_bHeatingOn := bHeatingOn;
END_GET
END_PROPERTY

PROPERTY P_nTempActual : UINT
GET
P_nTempActual := nTempActual;
END_GET
END_PROPERTY

PROPERTY P_nPidKi : UINT
SET
nPidKi := P_nPidKi;
END_SET
GET
P_nPidKi := nPidKi;
END_GET
END_PROPERTY

PROPERTY P_nTempSetpoint : USINT
SET
nTempSetpoint := P_nTempSetpoint;
END_SET
GET
P_nTempSetpoint := nTempSetpoint;
END_GET
END_PROPERTY

PROPERTY P_nPidKd : UINT
GET
P_nPidKd := nPidKd;
END_GET
SET
nPidKd := P_nPidKd;
END_SET
END_PROPERTY

PROPERTY P_bResetVialDetect : BOOL
SET
bResetVialDetect := P_bResetVialDetect;
END_SET
GET
P_bResetVialDetect := bResetVialDetect;
END_GET
END_PROPERTY

PROPERTY P_nPidTa : USINT
GET
P_nPidTa := nPidTa;
END_GET
SET
nPidTa := P_nPidTa;
END_SET
END_PROPERTY

PROPERTY P_bTempCutoff : BOOL
GET
P_bTempCutoff := bTempCutoff;
END_GET
END_PROPERTY

PROPERTY P_nPidKp : UINT
GET
P_nPidKp := nPidKp;
END_GET
SET
nPidKp := P_nPidKp;
END_SET
END_PROPERTY

PROPERTY P_bVialDetected : BOOL
GET
P_bVialDetected := bVialDetected;
END_GET
END_PROPERTY

END_FUNCTION_BLOCK

// ---- Hardware/Reactor/FB_ReactDriveInit.TcPOU
FUNCTION_BLOCK FB_ReactDriveInit
VAR_INPUT
	pDriveRef 	: POINTER TO FB_HwRefReactDrive;
	bExecute	: BOOL; 
END_VAR
VAR_OUTPUT
	bBusy		: BOOL;
	bError		: BOOL;
	nErrorId	: ERRORID;	
END_VAR
VAR
	fbSdoWrite	: FB_SDO_WRITE;
	fbPower		: FB_CANOpenMotionPower;
	nState		: USINT;
	nStateNext	: USINT;
	tmrTimeout	: TON;
	
	eCurrentDrive	: E_ReactDrive;
	
	nStateA 		: USINT;
	nStateANext 	: USINT;

	dwSdoIndex 		: DWORD;
	dwSdoSubIndex 	: DWORD;
	dwSdoDataLength : DWORD;
	nSdoDataValue 	: DINT;
END_VAR

VAR CONSTANT
	//Objekt-Indiezes
	cSdoIdxSwitchPara	: ARRAY[1..3] OF DWORD := [16#2005,16#2205,16#2405];
	cSdoIdxMaxCurrent	: ARRAY[1..3] OF DWORD := [16#2003,16#2203,16#2403];
	cSdoIdxHoldCurrent	: ARRAY[1..3] OF DWORD := [16#2004,16#2204,16#2404];
	cSdoIdxPulseDivisor	: ARRAY[1..3] OF DWORD := [16#2086,16#2286,16#2486];
	cSdoIdxPosWindow	: ARRAY[1..3] OF DWORD := [16#6067,16#6867,16#7067];
	cSdoIdxHomingMethod	: ARRAY[1..3] OF DWORD := [16#6098,16#6898,16#7098];
	cSdoIdxHomingSpeeds	: ARRAY[1..3] OF DWORD := [16#6099,16#6899,16#7099];
	cSdoIdxMoveSpeed	: ARRAY[1..3] OF DWORD := [16#6081,16#6881,16#7081];
	//Values
	cMaxCurrent			: ARRAY[1..3] OF DINT := [130,140,130];
	cHoldCurrent		: ARRAY[1..3] OF DINT := [32,32,32];
	cHomingSpeedFast	: ARRAY[1..3] OF DINT := [200,200,150];
	cHomingSpeedSlow	: ARRAY[1..3] OF DINT := [20,20,20];
	cHomingMethod		: ARRAY[1..3] OF DINT := [21,21,21];
	//cMoveSpeed			: ARRAY[1..3] OF DINT := [1500,1000,500];
	cGear				: ARRAY[1..3] OF REAL := [12.8,12.8,25.6];
END_VAR

IF bExecute THEN
	bBusy := TRUE;
	tmrTimeout();
	IF tmrTimeout.Q THEN
		bError := TRUE;
		bBusy := FALSE;
		nState := 99;
	END_IF
	
	CASE nState OF
		0:	pDriveRef^.bIsInit := FALSE;
			//Clamp
			eCurrentDrive := E_ReactDrive.Clamp;
			pDriveRef^.eCurrentState[1] := E_OpClState.UNDEFINED; 
			nState := 60;
			nStateNext := 1;
			
		1:	//Cover Vertikal
			eCurrentDrive := E_ReactDrive.CoverVerti;
			pDriveRef^.eCurrentState[2] := E_OpClState.UNDEFINED;
			nState := 60;
			nStateNext := 2;

		2:	//Cover Horizontal
			eCurrentDrive := E_ReactDrive.CoverHoriz;
			pDriveRef^.eCurrentState[3] := E_OpClState.UNDEFINED;
			nState := 60;
			nStateNext := 80;
		
		60:	//Prepare
			A_Prepare();
			IF nStateA >= 80 THEN
				IF nStateA >= 99 THEN
					bError := TRUE;
					bBusy := FALSE;
					nState := 99;
				ELSE
					nState := 61;
				END_IF
				nStateA := 0;
			END_IF
		
		61:	//PowerOn
			fbPower(pControl:= ADR(pDriveRef^.nControl[eCurrentDrive]), pStatus:= ADR(pDriveRef^.nStatus[eCurrentDrive]), bExecute:= TRUE);
			IF NOT 	fbPower.bBusy THEN
				IF fbPower.bError THEN
					nState := 99;
				ELSE
					nState := 62;
				END_IF
				fbPower(bExecute:= FALSE);
			END_IF		
		
		62:	//Init
			A_Init();
			IF nStateA >= 80 THEN
				IF nStateA >= 99 THEN
					nState := 99;
				ELSE
					nState := nStateNext;
					pDriveRef^.eCurrentState[eCurrentDrive] := E_OpClState.Open;
					IF nState = 80 THEN
						pDriveRef^.bIsInit := TRUE;
					END_IF
				END_IF
				nStateA := 0;
			END_IF
			
		70:	//Abbrechen
			//Das aktuelle Drive stoppen!
			nStateA := 70;
			A_Init();
			IF nStateA >= 80 THEN
				IF nStateA >= 99 THEN
					nState := 99;
				ELSE
					nState := 80;
				END_IF
				nStateA := 0;
			END_IF
		
		80:	//Ready
			bBusy := FALSE;
		
	END_CASE
ELSE
	fbPower(bExecute:= FALSE);
	tmrTimeout(IN:=FALSE);
	bError := FALSE;
	nErrorId := 0;
	nState := 0;
	nStateA := 0;
END_IF

ACTION A_Prepare:
CASE nStateA OF
	0:	//Errorbit gesetzt?
			IF pDriveRef^.nStatus[eCurrentDrive].3 THEN //Error zurücksetzen
				pDriveRef^.nControl[eCurrentDrive] := 153;
			ELSE
				pDriveRef^.nControl[eCurrentDrive] := 0;
				nStateA := 1;
			END_IF
			
	1:	//SwitchParameters setzen (keine Endlagen verwenden)
		dwSdoIndex := cSdoIdxSwitchPara[eCurrentDrive];
		dwSdoSubIndex := 0;
		dwSdoDataLength := 4;
		nSdoDataValue := 3; //keien Endlagen vewenden
		nStateANext := 2;
		nStateA := 60; //Sdo senden
		
	2:	//MaxCurrent setzen
		dwSdoIndex := cSdoIdxMaxCurrent[eCurrentDrive];
		dwSdoSubIndex := 0;
		dwSdoDataLength := 1;
		nSdoDataValue := cMaxCurrent[eCurrentDrive];
		nStateANext := 3;
		nStateA := 60; //Sdo senden
	
	3:	//HoldCurrent setzen
		dwSdoIndex := cSdoIdxHoldCurrent[eCurrentDrive];
		dwSdoSubIndex := 0;
		dwSdoDataLength := 1;
		nSdoDataValue := cHoldCurrent[eCurrentDrive];
		nStateANext := 4;
		nStateA := 60; //Sdo senden
	
	4:	//Homing Fast-Speed setzen
		dwSdoIndex := cSdoIdxHomingSpeeds[eCurrentDrive];
		dwSdoSubIndex := 1;
		dwSdoDataLength := 4;
		nSdoDataValue := cHomingSpeedFast[eCurrentDrive];
		nStateANext := 5;
		nStateA := 60; //Sdo senden
		
	5:	//Homing Slow-Speed setzen
		dwSdoIndex := cSdoIdxHomingSpeeds[eCurrentDrive];
		dwSdoSubIndex := 2;
		dwSdoDataLength := 4;
		nSdoDataValue := cHomingSpeedSlow[eCurrentDrive];
		nStateANext := 6;
		nStateA := 60; //Sdo senden		
		
	6:	//Pulse-Divisor setzen
		dwSdoIndex := cSdoIdxPulseDivisor[eCurrentDrive];
		dwSdoSubIndex := 0;
		dwSdoDataLength := 1;
		nSdoDataValue := 1;
		nStateANext := 7;
		nStateA := 60; //Sdo senden
		
	7:	//Position-Windows setzen
		dwSdoIndex := cSdoIdxPosWindow[eCurrentDrive];
		dwSdoSubIndex := 0;
		dwSdoDataLength := 4;
		nSdoDataValue := 100;
		nStateANext := 8;
		nStateA := 60; //Sdo senden		

	8:	//Move-Speed setzen
		dwSdoIndex := cSdoIdxMoveSpeed[eCurrentDrive];
		dwSdoSubIndex := 0;
		dwSdoDataLength := 4;
		nSdoDataValue := pDriveRef^.nMotorSpeed[eCurrentDrive];
		nStateANext := 9;
		nStateA := 60; //Sdo senden

	9:	//Homing Method setzen
		dwSdoIndex := cSdoIdxHomingMethod[eCurrentDrive];
		dwSdoSubIndex := 0;
		dwSdoDataLength := 1;
		nSdoDataValue := cHomingMethod[eCurrentDrive];
		nStateANext := 80;
		nStateA := 60; //Sdo senden		
		
	60:	//Send SDO
		fbSdoWrite(sADSNetID:= pDriveRef^.stAdsAdress.sNetId,nPortNr:= pDriveRef^.stAdsAdress.nPort, 
					nIndex:= dwSdoIndex, nSubIndex:= dwSdoSubIndex, nDataLength:= dwSdoDataLength,
					 nData:= nSdoDataValue, bExecute:= TRUE);
		IF NOT fbSdoWrite.bBusy THEN
			IF fbSdoWrite.bError THEN
				nErrorId := fbSdoWrite.nAdsErrorId;
				nStateA := 99;
			ELSE
				nStateA := nStateANext;
			END_IF
			fbSdoWrite(bExecute:= FALSE);
		END_IF
END_CASE
END_ACTION

METHOD M_Stop
VAR_INPUT
END_VAR
IF bBusy AND nState < 70 THEN
	nState := 70;	
END_IF
END_METHOD

ACTION A_Init:
CASE nStateA OF
	0:	
		pDriveRef^.nOpMode[eCurrentDrive] := 6;
		nStateA := 1;
		
	1: 
		IF pDriveRef^.nCurrentOpMode[eCurrentDrive] = 6 THEN
			pDriveRef^.nControl[eCurrentDrive] := 31;
			nStateA := 2;
		END_IF
		
	2:
		IF (pDriveRef^.nStatus[eCurrentDrive] AND 16#1400) = 16#1400 THEN
			pDriveRef^.nControl[eCurrentDrive] := 15;
			nStateA := 80;
		END_IF
		
	70:	//Abbrechen
		pDriveRef^.nControl[eCurrentDrive] := 15;
		nStateA := 80;
END_CASE
END_ACTION

END_FUNCTION_BLOCK

// ---- Hardware/Reactor/FB_ReactDriveMove.TcPOU
FUNCTION_BLOCK FB_ReactDriveMove
VAR_INPUT
	pDriveRef 	: POINTER TO FB_HwRefReactDrive;
	eDrive		: E_ReactDrive;
	eOpClCtrl	: E_OpClCtrl;
	bExecute	: BOOL; 
END_VAR
VAR_OUTPUT
	bBusy		: BOOL;
	bError		: BOOL;
	nErrorId	: ERRORID;	
END_VAR
VAR
	nState	: USINT;
END_VAR
VAR CONSTANT
	cGear	: ARRAY[1..3] OF REAL := [12.8, 12.8, 25.6];
END_VAR

IF bExecute THEN
	IF NOT pDriveRef^.bIsInit THEN
		nErrorId := E_ErrorIdCmd.ERRORID_DeviceNotInitialized;
		bError := TRUE;
		RETURN;
	END_IF

	pDriveRef^.eCurrentState[eDrive] := E_OpClState.UNDEFINED;
	IF pDriveRef^.nStatus[eDrive].3 THEN //Error
		bBusy := FALSE;
		bError := TRUE;
		RETURN;
	END_IF	

	IF nState = 0 THEN	//PP-Mode einstellen
		bBusy := TRUE;
		IF pDriveRef^.nCurrentOpMode[eDrive] <> 1 THEN
			pDriveRef^.nOpMode[eDrive] := 1;
		ELSE
			nState := 1;
			pDriveRef^.nControl[eDrive] := 15;
		END_IF
	END_IF
	
	IF nState = 1 THEN
		IF eOpClCtrl = E_OpClCtrl.Open THEN
			pDriveRef^.nTargetPos[eDrive] := 0;
		ELSE
			pDriveRef^.nTargetPos[eDrive] := REAL_TO_DINT(DINT_TO_REAL(pDriveRef^.nClosedPosition[eDrive]) * cGear[eDrive]);
		END_IF
		
		nState := 2;
	ELSIF nState = 2 THEN
		pDriveRef^.nControl[eDrive] := 31;
		nState := 3;
	ELSIF nState = 3 THEN
		IF pDriveRef^.nStatus[eDrive].12 THEN  //Setpoint ACK
			pDriveRef^.nControl[eDrive] := 15;
			nState := 4;
		END_IF
	ELSIF nState = 4 THEN
		IF pDriveRef^.nStatus[eDrive].10 THEN //TargetReached
			IF eOpClCtrl = E_OpClCtrl.Open THEN
				pDriveRef^.eCurrentState[eDrive] := E_OpClState.Open;
			ELSE
				pDriveRef^.eCurrentState[eDrive] := E_OpClState.Closed;
			END_IF
			bBusy := FALSE;
		END_IF
	END_IF
ELSE
	bError := FALSE;
	nErrorId := 0;
	nState := 0;
END_IF

END_FUNCTION_BLOCK

// ---- Objects/Tools/FB_FlipTubeHandler.TcPOU
FUNCTION_BLOCK FB_FlipTubeHandler EXTENDS FB_MzTool
VAR_INPUT
END_VAR
VAR_OUTPUT
END_VAR

SUPER^();	//FB_MzTool aufrufen

aObjProcData[nNotifyId] := stProcessData;

ACTION A_Reset:
//Ist noch eine Aktion aktiv?
IF nStateA_ResetSpec = 0 THEN 
	nStateA_ResetSpec := 80;
END_IF

SUPER^.A_Reset();
END_ACTION

METHOD FB_init : BOOL
VAR_INPUT
	bInitRetains : BOOL; // if TRUE, the retain variables are initialized (warm start / cold start)
	bInCopyCode : BOOL;  // if TRUE, the instance afterwards gets moved into the copy code (online change)
END_VAR
eObjectType := E_ObjectType.OBJECTTYPE_FlipTubeHandler;
eObjectGroup := E_ObjectGroup.OBJECTGROUP_MzTool OR E_ObjectGroup.OBJECTGROUP_Device;
END_METHOD

METHOD M_AddChild : ERRORID
VAR_INPUT
	pObject : POINTER TO FB_Object;
	nSlotNr	: UINT;
	nIndex 	: INT;
END_VAR
//Der Fliptube-Handler kann nur einen Exposure aufnehmen
IF pObject > 0 AND_THEN pObject^.P_eObjectType = E_ObjectType.OBJECTTYPE_Exposure THEN
	M_AddChild := SUPER^.M_AddChild(pObject,nSlotNr,nIndex);
ELSE
	M_AddChild := E_ErrorIdObjMgmt.ERRORID_InvalidParentObject;
END_IF
END_METHOD

METHOD M_CheckAction : ERRORID
VAR_INPUT
	refActionData 	: REFERENCE TO ST_ActionData;
	pCorrelObject	: POINTER TO FB_Object;
END_VAR
IF refActionData.eAction <> E_Action.ACTION_OpenCloseFlipTube THEN
	M_CheckAction := SUPER^.M_CheckAction(refActionData, pCorrelObject);
END_IF
END_METHOD

END_FUNCTION_BLOCK

// ---- Objects/Tools/FB_Luer.TcPOU
FUNCTION_BLOCK FB_Luer EXTENDS FB_GCodeTool  IMPLEMENTS I_UsingDryPad
VAR_INPUT
END_VAR
VAR_OUTPUT
END_VAR
VAR
	//SpecProperties
	nDiluterObjId		: UINT;
	nDiluterObjId2		: UINT;
	pDiluter			: POINTER TO FB_Diluter;
	pDiluter2			: POINTER TO FB_Diluter;
	nDrypadArea			: USINT;
	tDryTime			: TIME;
	pPneuChannelSyntGas	: POINTER TO FB_PneuChannelRef;
	
	nValveNrSynthGas	: USINT;
	nValveNrDiluter		: USINT;
	nValveNrLuer		: USINT;
	rDockOffset			: REAL;
	
	nDispFlowFix		: DINT;
	
	//****************************************Aktionvariablen****************************************************
	
	stActionDataSpec	: ST_ActionData;
	
	//Action: "Aspirate"
	bAspirate			: BOOL;
	nStateA_Aspirate	: USINT;
	nQuantity			: DINT;
	nFlow				: DINT;
	
	//Action: "Dispense"
	bDispense			: BOOL;
	nStateA_Dispense	: USINT;
	bEndless			: BOOL;
	
	//Action: "Mix"
	bMix				: BOOL;
	nStateA_Mix			: USINT;
	nFlowAsp			: DINT;
	nFlowDisp			: DINT;
	nMixRepeats			: UINT;
	nCurrMixRepeats		: UINT;
	tMixDelay1			: TIME; //Delay zwischen Asp und Disp
	tMixDelay2			: TIME; //Delay nach jedem Zyklus
	timerMix			: TON;
	
	//Action: "Eject"
	bEject				: BOOL;
	nStateA_Eject		: USINT;
	fbMultiZTipEjector	: FB_MultiZTipEjector;
	
	//Action: "SetPressure"
	bSetPress			: BOOL;
	fbSetPress			: FB_SetPressure;
	
	//Action: "SwitchPressure"
	bSwitchPress		: BOOL;			
	nStateA_SwitchPress	: USINT;		//State von A_SwitchPress()
	eSwitchPressCtrl	: E_PressCtrl;
	tPressTime			: TIME;			//nach dieser Zeit Ventil automatisch wieder zu
	timerPress			: TON;			//Timer für Öffnungszeit Druckventil 	
END_VAR

IF eCurrentState = E_MachineState.MACHINESTATE_Active THEN
	
	IF bAspirate THEN
		A_Aspirate();
		IF nStateA_Aspirate >= 80 THEN
			IF nStateA_Aspirate >= 99 THEN
				bError := TRUE;	
			END_IF
			bAspirate := FALSE;
			nStateA_Aspirate := 0;
			M_RemoveListEntry(nSearchValue:= E_Action.ACTION_Aspirate);
		END_IF
	END_IF

	IF bDispense THEN
		A_Dispense();
		IF nStateA_Dispense >= 80 THEN
			IF nStateA_Dispense >= 99 THEN
				bError := TRUE;	
			END_IF
			bDispense := FALSE;
			nStateA_Dispense := 0;
			M_RemoveListEntry(nSearchValue:= E_Action.ACTION_Dispense);
		END_IF
	END_IF
	
	IF bMix THEN
		A_Mix();
		IF nStateA_Mix >= 80 THEN
			IF nStateA_Mix >= 99 THEN
				stError.Cmd := E_Action.ACTION_Mix;
				fbErrorList.M_Add(stError);
				bError := TRUE;	
			END_IF
			bMix := FALSE;
			nStateA_Mix := 0;
			M_RemoveListEntry(nSearchValue:= E_Action.ACTION_Mix);
		END_IF
	END_IF
	
	IF bEject THEN
		A_Eject();
		IF nStateA_Eject >= 80 THEN
			IF nStateA_Eject >= 99 THEN
				bError := TRUE;	
			END_IF
			bEject := FALSE;
			nStateA_Eject := 0;
			M_RemoveListEntry(nSearchValue:= E_Action.ACTION_Eject);
		END_IF
	END_IF
	
	IF bSetPress THEN
		fbSetPress(pPneuChannelRef:= pPneuChannelSyntGas);
		IF NOT fbSetPress.bBusy THEN
			IF fbSetPress.bError THEN
				bError := TRUE;
				stError.ErrorId := fbSetPress.nErrorId;
				stError.POU := E_POU.POU_FB_Luer;
				fbErrorList.M_Add(stError);
			END_IF
			bSetPress := FALSE;
			fbSetPress(pPneuChannelRef:= pPneuChannelSyntGas, bExecute:= FALSE);
			M_RemoveListEntry(nSearchValue:= E_Action.ACTION_SetPressure);
		END_IF
	END_IF	
	
	IF bSwitchPress THEN	//Kartuschendruck einstellen und Ein-bzw. Aus schalten 
		A_SwitchPress();
		IF nStateA_SwitchPress >= 80 THEN
			IF nStateA_SwitchPress >= 99 THEN
				bError := TRUE;
			END_IF
			bSwitchPress := FALSE;
			nStateA_SwitchPress := 0;
			M_RemoveListEntry(nSearchValue:= E_Action.ACTION_SwitchPressure);
		END_IF
	END_IF	

END_IF

SUPER^();	//FB_MzTool aufrufen

//Prozessdaten aktualisieren
IF pPneuChannelSyntGas > 0 THEN
	stProcessData.n32Data[7] := pPneuChannelSyntGas^.P_nCurrentPressure;
END_IF

IF nValveNrSynthGas > 0 THEN
	IF aValves[nValveNrSynthGas].bDigiOut1 THEN
		stProcessData.n32Data[8] := E_PressCtrl.PRESSCTRL_PressOn;
	ELSE
		stProcessData.n32Data[8] := E_PressCtrl.PRESSCTRL_Off;
	END_IF
END_IF

aObjProcData[nNotifyId] := stProcessData;

ACTION A_Aspirate:
IF pDiluter^.P_bError THEN
	stError.ErrorId := pDiluter^.P_nErrorId;
	stError.POUState := nStateA_Aspirate;
	nStateA_Aspirate := 99;
END_IF

CASE nStateA_Aspirate OF
	0:	
		M_SwitchValveDiluter(TRUE);
		M_SwitchValveLuer(TRUE);
		
		MEMSET(ADR(stActionDataSpec),0,SIZEOF(stActionDataSpec));
		stActionDataSpec.eAction := E_Action.ACTION_DilPump;
		stActionDataSpec.aParams[1] := E_DilPumpMode.MODE_Suck;
		stActionDataSpec.aParams[2] := nQuantity; 
		stActionDataSpec.aParams[3] := nFlow;
		//stActionDataSpec.aParams[4] := 2000; //ReloadSpeed wird von DilConfig übernommen
		//stActionDataSpec.aParams[5] := 3; //Valve-Position für Pump
		//stActionDataSpec.aParams[6] := 4; //Valve-Position für Reload (in Waste)

		stError.ErrorId := pDiluter^.M_ExeAction(stActionDataSpec);
		IF stError.ErrorId > 0 THEN
			stError.POUState := nStateA_Aspirate;
			nStateA_Aspirate := 99;
		ELSE
			nStateA_Aspirate := 1;	
		END_IF
		
	1:	//Warten bis Aspiration fertig
		IF NOT pDiluter^.M_GetActionBusy(E_Action.ACTION_DilPump) THEN
			M_SwitchValveDiluter(FALSE);
			M_SwitchValveLuer(FALSE);
			nStateA_Aspirate := 80;
		END_IF
		
	70:	//Abbrechen
		MEMSET(ADR(stActionDataSpec),0,SIZEOF(stActionDataSpec));
		stActionDataSpec.eAction := E_Action.ACTION_Stop;
		pDiluter^.M_ExeAction(stActionDataSpec);
		nStateA_Aspirate := 71;
		
	71:	
		IF NOT pDiluter^.P_bBusy THEN
			M_SwitchValveDiluter(FALSE);
			M_SwitchValveLuer(FALSE);
			nStateA_Aspirate := 80;
		END_IF
END_CASE

//Errorhandling
IF nStateA_Aspirate = 99 THEN
	stError.Cmd := E_Action.ACTION_Aspirate;
	stError.POU := E_POU.POU_FB_Luer;
	stError.POUAction := E_POUACT.POUACT_A_Aspirate;
	fbErrorList.M_Add(stError);
END_IF
END_ACTION

ACTION A_Dispense:
IF pDiluter^.P_bError THEN
	stError.ErrorId := pDiluter^.P_nErrorId;
	stError.POUState := nStateA_Dispense;
	nStateA_Dispense := 99;
END_IF

CASE nStateA_Dispense OF
	0:
		M_SwitchValveDiluter(TRUE);
		M_SwitchValveLuer(TRUE);
	
		MEMSET(ADR(stActionDataSpec),0,SIZEOF(stActionDataSpec));
		stActionDataSpec.eAction := E_Action.ACTION_DilPump;
		stActionDataSpec.aParams[1] := E_DilPumpMode.MODE_Press;
		stActionDataSpec.aParams[2] := nQuantity; 
		stActionDataSpec.aParams[3] := nFlow;
		
		stActionDataSpec.aParams[7] := BOOL_TO_DINT(bEndless);
		bEndless := FALSE;
		
		stError.ErrorId := pDiluter^.M_ExeAction(stActionDataSpec);
		IF stError.ErrorId > 0 THEN
			stError.POUState := nStateA_Dispense;
			nStateA_Dispense := 99;
		ELSE
			nStateA_Dispense := 1;	
		END_IF
		
	1:	//Warten bis Dispensen fertig
		IF NOT pDiluter^.M_GetActionBusy(E_Action.ACTION_DilPump) THEN
			M_SwitchValveDiluter(FALSE);
			M_SwitchValveLuer(FALSE);
			nStateA_Dispense := 80;
		END_IF
		
	70:	//Abbrechen
		MEMSET(ADR(stActionDataSpec),0,SIZEOF(stActionDataSpec));
		stActionDataSpec.eAction := E_Action.ACTION_Stop;
		
		pDiluter^.M_ExeAction(stActionDataSpec);
		nStateA_Dispense := 71;
		
	71:	
		IF NOT pDiluter^.P_bBusy THEN
			M_SwitchValveDiluter(FALSE);
			M_SwitchValveLuer(FALSE);
			nStateA_Dispense := 80;
		END_IF
END_CASE

//Errorhandling
IF nStateA_Dispense = 99 THEN
	stError.Cmd := E_Action.ACTION_Dispense;
	stError.POU := E_POU.POU_FB_Luer;
	stError.POUAction := E_POUACT.POUACT_A_Dispense;
	fbErrorList.M_Add(stError);
END_IF
END_ACTION

ACTION A_Eject:
fbMultiZTipEjector(pfbZAxisRef:= pZAxisRef, bExecute:= TRUE);

IF NOT fbMultiZTipEjector.bBusy THEN
	IF fbMultiZTipEjector.bError THEN
		stError.Cmd := E_Action.ACTION_Eject;
		stError.ErrorId := fbMultiZTipEjector.nErrorId;
		stError.POUState := nStateA_Eject;
		stError.POU := E_POU.POU_FB_Luer;
		stError.POUAction := E_POUACT.POUACT_A_Eject;
		fbErrorList.M_Add(stError);
		nStateA_Eject := 99;
	ELSE
		nStateA_Eject := 80;
	END_IF
	fbMultiZTipEjector(bExecute:= FALSE);
END_IF
END_ACTION

ACTION A_Mix:
IF pDiluter^.P_bError THEN
	stError.ErrorId := pDiluter^.P_nErrorId;
	stError.POUState := nStateA_Mix;
	nStateA_Mix := 99;
END_IF

CASE nStateA_Mix OF
	0:	//Aspirieren
	
		M_SwitchValveDiluter(TRUE);
		M_SwitchValveLuer(TRUE);
	
		MEMSET(ADR(stActionDataSpec),0,SIZEOF(stActionDataSpec));
		stActionDataSpec.eAction := E_Action.ACTION_DilPump;
		stActionDataSpec.aParams[1] := E_DilPumpMode.MODE_Suck;
		stActionDataSpec.aParams[2] := nQuantity; 
		stActionDataSpec.aParams[3] := nFlowAsp;
		
		stError.ErrorId := pDiluter^.M_ExeAction(stActionDataSpec);
		IF stError.ErrorId > 0 THEN
			stError.POUState := nStateA_Mix;
			nStateA_Mix := 99;
		ELSE
			nStateA_Mix := 1;	
		END_IF
		
	1:	//Aspirieren fertig?
		IF NOT pDiluter^.M_GetActionBusy(E_Action.ACTION_DilPump) THEN
			timerMix(IN:= TRUE, PT:= tMixDelay1);
			nStateA_Mix := 2;	
		END_IF
		
	2:	//Timer?
		timerMix();
		IF timerMix.Q THEN
			timerMix(IN:= FALSE);
			nStateA_Mix := 3;
		END_IF
		
	3:	//Dispensen
		MEMSET(ADR(stActionDataSpec),0,SIZEOF(stActionDataSpec));
		stActionDataSpec.eAction := E_Action.ACTION_DilPump;
		stActionDataSpec.aParams[1] := E_DilPumpMode.MODE_Press;
		stActionDataSpec.aParams[2] := nQuantity; 
		stActionDataSpec.aParams[3] := nFlowDisp;
		
		stError.ErrorId := pDiluter^.M_ExeAction(stActionDataSpec);
		IF stError.ErrorId > 0 THEN
			stError.POUState := nStateA_Mix;
			nStateA_Mix := 99;
		ELSE
			nStateA_Mix := 4;
		END_IF
		
	4:	//Dispensen fertig?
		IF NOT pDiluter^.M_GetActionBusy(E_Action.ACTION_DilPump) THEN
			nCurrMixRepeats := nCurrMixRepeats + 1;
			IF nCurrMixRepeats = nMixRepeats THEN
				M_SwitchValveDiluter(FALSE);
				M_SwitchValveLuer(FALSE);
				nStateA_Mix := 80;
			ELSE
				timerMix(IN:= TRUE, PT:= tMixDelay2);
				nStateA_Mix := 5;
			END_IF
		END_IF
		
	5:	//Timer?
		timerMix();
		IF timerMix.Q THEN
			timerMix(IN:= FALSE);
			nStateA_Mix := 0;
		END_IF

	70:	//Abbrechen
		timerMix(IN:= FALSE);
		MEMSET(ADR(stActionDataSpec),0,SIZEOF(stActionDataSpec));
		stActionDataSpec.eAction := E_Action.ACTION_Stop;
		pDiluter^.M_ExeAction(stActionDataSpec);
		nStateA_Mix := 71;
		
	71:	IF NOT pDiluter^.P_bBusy THEN
			M_SwitchValveDiluter(FALSE);
			M_SwitchValveLuer(FALSE);
			nStateA_Mix := 80;
		END_IF		
END_CASE

//Errorhandling
IF nStateA_Mix = 99 THEN
	stError.Cmd := E_Action.ACTION_Mix;
	stError.POU := E_POU.POU_FB_PassivPip;
	stError.POUAction := E_POUACT.POUACT_A_Mix;
	fbErrorList.M_Add(stError);
END_IF
END_ACTION

ACTION A_Reset:
//Ist noch eine Aktion aktiv?
IF nStateA_ResetSpec = 0 THEN 

	IF bSetPress THEN
		bSetPress := FALSE;
		fbSetPress(bExecute:= FALSE, pPneuChannelRef:= pPneuChannelSyntGas);
	END_IF	

	IF bAspirate THEN
		bAspirate := FALSE;
		nStateA_Aspirate := 0;
	END_IF

	IF bDispense THEN
		bDispense := FALSE;
		nStateA_Dispense := 0;
	END_IF
	
	IF bEject THEN
		bEject := FALSE;
		nStateA_Eject := 0;
	END_IF
	
	nStateA_ResetSpec := 80;
END_IF

SUPER^.A_Reset();
END_ACTION

ACTION A_Stop:
IF nStateA_Stop = 0 THEN
	
	IF bAspirate AND nStateA_Aspirate < 70 THEN
		nStateA_Aspirate := 70;
	END_IF
	
	IF bDispense AND nStateA_Dispense < 70 THEN
		nStateA_Dispense := 70;
	END_IF
	
	IF bMix AND nStateA_Mix < 70 THEN
		nStateA_Mix := 70;
	END_IF
	
	IF bSetPress THEN
		fbSetPress(bExecute:= FALSE, pPneuChannelRef:= pPneuChannelSyntGas);
	END_IF
	
	IF bSwitchPress AND nStateA_SwitchPress < 70 THEN
		nStateA_SwitchPress := 70;
	END_IF	
	
	nStateA_Stop := 1;
END_IF

SUPER^.A_Stop();
END_ACTION

ACTION A_SwitchPress:
CASE nStateA_SwitchPress OF
	0:	//Ventil Einschalten
		//Das ValveLuer muss ebenfalls ausgeschalten werden
		IF eSwitchPressCtrl = E_PressCtrl.PRESSCTRL_PressOn THEN
			M_SwitchValveLuer(FALSE);
			M_SwitchValveSynthGas(TRUE);
		END_IF
	
		//Timer starten
		IF tPressTime = T#0S THEN
			nStateA_SwitchPress := 80;
			RETURN;	
		END_IF
		
		timerPress(IN:= FALSE);
		timerPress(IN:= TRUE, PT:= tPressTime);
		nStateA_SwitchPress := 1;
		
	1:	//Warten bis Zeitabgelaufen
		timerPress();
		IF timerPress.Q THEN
			timerPress(IN:= FALSE);
			M_SwitchValveSynthGas(FALSE);
			nStateA_SwitchPress := 80;
		END_IF
		
	70:	//Abbrechen
		timerPress(IN:= FALSE);
		M_SwitchValveSynthGas(FALSE);
		nStateA_SwitchPress := 80;
END_CASE
END_ACTION

METHOD FB_init : BOOL
VAR_INPUT
	bInitRetains : BOOL; // if TRUE, the retain variables are initialized (warm start / cold start)
	bInCopyCode : BOOL;  // if TRUE, the instance afterwards gets moved into the copy code (online change)
END_VAR
eObjectType := E_ObjectType.OBJECTTYPE_Luer;
eObjectGroup := E_ObjectGroup.OBJECTGROUP_MzTool OR E_ObjectGroup.OBJECTGROUP_Device;
END_METHOD

METHOD M_AddChild : ERRORID
VAR_INPUT
	pObject : POINTER TO FB_Object;
	nSlotNr	: UINT;
	nIndex 	: INT;
END_VAR
//Der Luer kann folgende Objekt-Typen aufnehmen
//Needle, Tip
IF pObject > 0 THEN
	IF pObject^.P_eObjectType = E_ObjectType.OBJECTTYPE_Needle OR
		pObject^.P_eObjectType = E_ObjectType.OBJECTTYPE_DummyTool OR
		pObject^.P_eObjectType = E_ObjectType.OBJECTTYPE_Tip THEN
		M_AddChild := SUPER^.M_AddChild(pObject,nSlotNr,nIndex);
	ELSE
		M_AddChild := E_ErrorIdObjMgmt.ERRORID_InvalidParentObject;
	END_IF
ELSE
	M_AddChild := E_ErrorIdObjMgmt.ERRORID_InvalidParentObject;
END_IF
END_METHOD

METHOD M_CancelAction
VAR_INPUT
	eAction : E_Action;
END_VAR
CASE eAction OF
	E_Action.ACTION_Aspirate:
		IF bAspirate AND nStateA_Aspirate < 70 THEN
			nStateA_Aspirate := 70;
		END_IF
	E_Action.ACTION_Dispense:
		IF bDispense AND nStateA_Dispense < 70 THEN
			nStateA_Dispense := 70;
		END_IF
	E_Action.ACTION_Mix:
		IF bMix AND nStateA_Mix < 70 THEN
			nStateA_Mix := 70;
		END_IF			
	E_Action.ACTION_SetPressure:
	IF bSetPress THEN
		fbSetPress(bExecute:= FALSE, pPneuChannelRef:= pPneuChannelSyntGas);
	END_IF
	E_Action.ACTION_SwitchPressure:
		IF bSwitchPress AND nStateA_SwitchPress < 70 THEN
			nStateA_SwitchPress := 70;
		END_IF	
ELSE
	SUPER^.M_CancelAction(eAction);
END_CASE
END_METHOD

METHOD M_CheckAction : ERRORID
VAR_INPUT
	refActionData 	: REFERENCE TO ST_ActionData;
	pCorrelObject	: POINTER TO FB_Object;
END_VAR

